(* CoDeSys 2.3.9.50 project: STP_PLC_arc.pro *)
(* Libraries: STANDARD.LIB 5.6.98 12:03:02 *)

(* Task configuration *)
TASK Standard (PRIORITY := 0, INTERVAL := T#10ms);
	STP
END_TASK

(* Global variable list: TwinCAT_Configuration *)
(* Generated automatically by TwinCAT - (read only) *)
VAR_CONFIG
	STP.LSL100A_MixerFloatSensor AT %IX276.0 : BOOL;	(*  ~ {LinkedWith:TIID^C6920 (EtherCAT)^ScadaRoom_KouplerUTP (EK1100)^ScadaRoom_KouplerFiber (EK1521)^InletWork_1(EK1501)^Term 5 (EL1809)^Channel 1^Input} *)
	STP.LSH100A_MixerFloatSensor AT %IX272.0 : BOOL;	(*  ~ {LinkedWith:TIID^C6920 (EtherCAT)^ScadaRoom_KouplerUTP (EK1100)^ScadaRoom_KouplerFiber (EK1521)^InletWork_1(EK1501)^Term 5 (EL1809)^Channel 2^Input} *)
	STP.LSH101A_EQFloatSensor AT %IX276.1 : BOOL;	(*  ~ {LinkedWith:TIID^C6920 (EtherCAT)^ScadaRoom_KouplerUTP (EK1100)^ScadaRoom_KouplerFiber (EK1521)^InletWork_1(EK1501)^Term 5 (EL1809)^Channel 3^Input} *)
	STP.LSHH101A_EQFloatSensor AT %IX276.2 : BOOL;	(*  ~ {LinkedWith:TIID^C6920 (EtherCAT)^ScadaRoom_KouplerUTP (EK1100)^ScadaRoom_KouplerFiber (EK1521)^InletWork_1(EK1501)^Term 5 (EL1809)^Channel 4^Input} *)
	STP.LSL101A_EQFloatSensor AT %IX256.1 : BOOL;	(*  ~ {LinkedWith:TIID^C6920 (EtherCAT)^ScadaRoom_KouplerUTP (EK1100)^ScadaRoom_KouplerFiber (EK1521)^InletWork_1(EK1501)^Term 5 (EL1809)^Channel 5^Input} *)
	STP.LSH105A1_StreamLineFlow AT %IX276.3 : BOOL;	(*  ~ {LinkedWith:TIID^C6920 (EtherCAT)^ScadaRoom_KouplerUTP (EK1100)^ScadaRoom_KouplerFiber (EK1521)^InletWork_1(EK1501)^Term 5 (EL1809)^Channel 6^Input} *)
	STP.LSHH105A2_StreamLineOverflow AT %IX276.4 : BOOL;	(*  ~ {LinkedWith:TIID^C6920 (EtherCAT)^ScadaRoom_KouplerUTP (EK1100)^ScadaRoom_KouplerFiber (EK1521)^InletWork_1(EK1501)^Term 5 (EL1809)^Channel 7^Input} *)
	STP.LSL103A_SBRFloatSensor AT %IX256.2 : BOOL;	(*  ~ {LinkedWith:TIID^C6920 (EtherCAT)^ScadaRoom_KouplerUTP (EK1100)^ScadaRoom_KouplerFiber (EK1521)^InletWork_1(EK1501)^Term 5 (EL1809)^Channel 8^Input} *)
	STP.LSHH103A_SBRFloatSensor AT %IX276.6 : BOOL;	(*  ~ {LinkedWith:TIID^C6920 (EtherCAT)^ScadaRoom_KouplerUTP (EK1100)^ScadaRoom_KouplerFiber (EK1521)^InletWork_1(EK1501)^Term 5 (EL1809)^Channel 9^Input} *)
	STP.LSH103A_SBRFloatSensor AT %IX276.5 : BOOL;	(*  ~ {LinkedWith:TIID^C6920 (EtherCAT)^ScadaRoom_KouplerUTP (EK1100)^ScadaRoom_KouplerFiber (EK1521)^InletWork_1(EK1501)^Term 5 (EL1809)^Channel 10^Input} *)
	STP.TMT01_FanStatus AT %IX276.7 : BOOL;	(*  ~ {LinkedWith:TIID^C6920 (EtherCAT)^ScadaRoom_KouplerUTP (EK1100)^ScadaRoom_KouplerFiber (EK1521)^InletWork_1(EK1501)^Term 5 (EL1809)^Channel 11^Input} *)
	STP.DP01_DoorPanelStatus AT %IX277.0 : BOOL;	(*  ~ {LinkedWith:TIID^C6920 (EtherCAT)^ScadaRoom_KouplerUTP (EK1100)^ScadaRoom_KouplerFiber (EK1521)^InletWork_1(EK1501)^Term 5 (EL1809)^Channel 12^Input} *)
	STP.LSD101A_EQFloatSensorDry AT %IX277.1 : BOOL;	(*  ~ {LinkedWith:TIID^C6920 (EtherCAT)^ScadaRoom_KouplerUTP (EK1100)^ScadaRoom_KouplerFiber (EK1521)^InletWork_1(EK1501)^Term 5 (EL1809)^Channel 13^Input} *)
	STP.LSD103A_SBRFloatSensorDry AT %IX277.2 : BOOL;	(*  ~ {LinkedWith:TIID^C6920 (EtherCAT)^ScadaRoom_KouplerUTP (EK1100)^ScadaRoom_KouplerFiber (EK1521)^InletWork_1(EK1501)^Term 5 (EL1809)^Channel 14^Input} *)
	STP.XV101A1_SolenoidValveSpray_OpenStat AT %IX277.3 : BOOL;	(*  ~ {LinkedWith:TIID^C6920 (EtherCAT)^ScadaRoom_KouplerUTP (EK1100)^ScadaRoom_KouplerFiber (EK1521)^InletWork_1(EK1501)^Term 6 (EL1809)^Channel 1^Input} *)
	STP.XV101A2_SolenoidValveSpray_OpenStat AT %IX277.4 : BOOL;	(*  ~ {LinkedWith:TIID^C6920 (EtherCAT)^ScadaRoom_KouplerUTP (EK1100)^ScadaRoom_KouplerFiber (EK1521)^InletWork_1(EK1501)^Term 6 (EL1809)^Channel 2^Input} *)
	STP.XV102A1_ContinuosValveWater_OpenStat AT %IX277.5 : BOOL;	(*  ~ {LinkedWith:TIID^C6920 (EtherCAT)^ScadaRoom_KouplerUTP (EK1100)^ScadaRoom_KouplerFiber (EK1521)^InletWork_1(EK1501)^Term 6 (EL1809)^Channel 3^Input} *)
	STP.XV100A1_GritRemovalValve_OpenStat AT %IX277.6 : BOOL;	(*  ~ {LinkedWith:TIID^C6920 (EtherCAT)^ScadaRoom_KouplerUTP (EK1100)^ScadaRoom_KouplerFiber (EK1521)^InletWork_1(EK1501)^Term 6 (EL1809)^Channel 5^Input} *)
	STP.XV100A2_GritRemovalValve_OpenStat AT %IX277.7 : BOOL;	(*  ~ {LinkedWith:TIID^C6920 (EtherCAT)^ScadaRoom_KouplerUTP (EK1100)^ScadaRoom_KouplerFiber (EK1521)^InletWork_1(EK1501)^Term 6 (EL1809)^Channel 6^Input} *)
	STP.PS101A1_Penstock_OpenStat AT %IX278.0 : BOOL;	(*  ~ {LinkedWith:TIID^C6920 (EtherCAT)^ScadaRoom_KouplerUTP (EK1100)^ScadaRoom_KouplerFiber (EK1521)^InletWork_1(EK1501)^Term 6 (EL1809)^Channel 7^Input} *)
	STP.PS101A2_Penstock_OpenStat AT %IX278.1 : BOOL;	(*  ~ {LinkedWith:TIID^C6920 (EtherCAT)^ScadaRoom_KouplerUTP (EK1100)^ScadaRoom_KouplerFiber (EK1521)^InletWork_1(EK1501)^Term 6 (EL1809)^Channel 8^Input} *)
	STP.PS101A1_Penstock_CloseStat AT %IX278.2 : BOOL;	(*  ~ {LinkedWith:TIID^C6920 (EtherCAT)^ScadaRoom_KouplerUTP (EK1100)^ScadaRoom_KouplerFiber (EK1521)^InletWork_1(EK1501)^Term 6 (EL1809)^Channel 9^Input} *)
	STP.PS101A2_Penstock_CloseStat AT %IX278.3 : BOOL;	(*  ~ {LinkedWith:TIID^C6920 (EtherCAT)^ScadaRoom_KouplerUTP (EK1100)^ScadaRoom_KouplerFiber (EK1521)^InletWork_1(EK1501)^Term 6 (EL1809)^Channel 10^Input} *)
	STP.XV101A1_SolenoidValveSpray_CloseStat AT %IX278.4 : BOOL;	(*  ~ {LinkedWith:TIID^C6920 (EtherCAT)^ScadaRoom_KouplerUTP (EK1100)^ScadaRoom_KouplerFiber (EK1521)^InletWork_1(EK1501)^Term 6 (EL1809)^Channel 11^Input} *)
	STP.XV101A2_SolenoidValveSpray_CloseStat AT %IX278.5 : BOOL;	(*  ~ {LinkedWith:TIID^C6920 (EtherCAT)^ScadaRoom_KouplerUTP (EK1100)^ScadaRoom_KouplerFiber (EK1521)^InletWork_1(EK1501)^Term 6 (EL1809)^Channel 12^Input} *)
	STP.XV102A1_ContinuosValveWater_CloseStat AT %IX278.6 : BOOL;	(*  ~ {LinkedWith:TIID^C6920 (EtherCAT)^ScadaRoom_KouplerUTP (EK1100)^ScadaRoom_KouplerFiber (EK1521)^InletWork_1(EK1501)^Term 6 (EL1809)^Channel 13^Input} *)
	STP.XV100A1_GritRemovalValve_CloseStat AT %IX278.7 : BOOL;	(*  ~ {LinkedWith:TIID^C6920 (EtherCAT)^ScadaRoom_KouplerUTP (EK1100)^ScadaRoom_KouplerFiber (EK1521)^InletWork_1(EK1501)^Term 6 (EL1809)^Channel 14^Input} *)
	STP.XV100A2_GritRemovalValve_CloseStat AT %IX279.0 : BOOL;	(*  ~ {LinkedWith:TIID^C6920 (EtherCAT)^ScadaRoom_KouplerUTP (EK1100)^ScadaRoom_KouplerFiber (EK1521)^InletWork_1(EK1501)^Term 6 (EL1809)^Channel 15^Input} *)
	STP.M101A1_EQMixer_OverloadStat AT %IX279.1 : BOOL;	(*  ~ {LinkedWith:TIID^C6920 (EtherCAT)^ScadaRoom_KouplerUTP (EK1100)^ScadaRoom_KouplerFiber (EK1521)^InletWork_1(EK1501)^Term 7 (EL1809)^Channel 1^Input} *)
	STP.M101A1_EQMixer_IncompleteStat AT %IX279.2 : BOOL;	(*  ~ {LinkedWith:TIID^C6920 (EtherCAT)^ScadaRoom_KouplerUTP (EK1100)^ScadaRoom_KouplerFiber (EK1521)^InletWork_1(EK1501)^Term 7 (EL1809)^Channel 2^Input} *)
	STP.M101A2_EQMixer_OverloadStat AT %IX279.3 : BOOL;	(*  ~ {LinkedWith:TIID^C6920 (EtherCAT)^ScadaRoom_KouplerUTP (EK1100)^ScadaRoom_KouplerFiber (EK1521)^InletWork_1(EK1501)^Term 7 (EL1809)^Channel 3^Input} *)
	STP.M101A2_EQMixer_IncompleteStat AT %IX279.4 : BOOL;	(*  ~ {LinkedWith:TIID^C6920 (EtherCAT)^ScadaRoom_KouplerUTP (EK1100)^ScadaRoom_KouplerFiber (EK1521)^InletWork_1(EK1501)^Term 7 (EL1809)^Channel 4^Input} *)
	STP.P101A1_EQPump_OverloadStat AT %IX4.0 : BOOL;	(*  ~ {LinkedWith:TIID^C6920 (EtherCAT)^ScadaRoom_KouplerUTP (EK1100)^ScadaRoom_KouplerFiber (EK1521)^InletWork_1(EK1501)^Term 7 (EL1809)^Channel 5^Input} *)
	STP.P101A1_EQPump_IncompleteStat AT %IX4.1 : BOOL;	(*  ~ {LinkedWith:TIID^C6920 (EtherCAT)^ScadaRoom_KouplerUTP (EK1100)^ScadaRoom_KouplerFiber (EK1521)^InletWork_1(EK1501)^Term 7 (EL1809)^Channel 6^Input} *)
	STP.P101A2_EQPump_OverloadStat AT %IX4.2 : BOOL;	(*  ~ {LinkedWith:TIID^C6920 (EtherCAT)^ScadaRoom_KouplerUTP (EK1100)^ScadaRoom_KouplerFiber (EK1521)^InletWork_1(EK1501)^Term 7 (EL1809)^Channel 7^Input} *)
	STP.P101A2_EQPump_IncompleteStat AT %IX4.3 : BOOL;	(*  ~ {LinkedWith:TIID^C6920 (EtherCAT)^ScadaRoom_KouplerUTP (EK1100)^ScadaRoom_KouplerFiber (EK1521)^InletWork_1(EK1501)^Term 7 (EL1809)^Channel 8^Input} *)
	STP.PS101A1_Penstock_TripStat AT %IX4.4 : BOOL;	(*  ~ {LinkedWith:TIID^C6920 (EtherCAT)^ScadaRoom_KouplerUTP (EK1100)^ScadaRoom_KouplerFiber (EK1521)^InletWork_1(EK1501)^Term 7 (EL1809)^Channel 9^Input} *)
	STP.PS101A2_Penstock_TripStat AT %IX4.5 : BOOL;	(*  ~ {LinkedWith:TIID^C6920 (EtherCAT)^ScadaRoom_KouplerUTP (EK1100)^ScadaRoom_KouplerFiber (EK1521)^InletWork_1(EK1501)^Term 7 (EL1809)^Channel 10^Input} *)
	STP.F101A1_FineScr_OverloadStat AT %IX4.6 : BOOL;	(*  ~ {LinkedWith:TIID^C6920 (EtherCAT)^ScadaRoom_KouplerUTP (EK1100)^ScadaRoom_KouplerFiber (EK1521)^InletWork_1(EK1501)^Term 8 (EL1809)^Channel 1^Input} *)
	STP.F101A2_FineScr_OverloadStat AT %IX4.7 : BOOL;	(*  ~ {LinkedWith:TIID^C6920 (EtherCAT)^ScadaRoom_KouplerUTP (EK1100)^ScadaRoom_KouplerFiber (EK1521)^InletWork_1(EK1501)^Term 8 (EL1809)^Channel 2^Input} *)
	STP.C102A_ScreeningConveyer_OverloadStat AT %IX5.0 : BOOL;	(*  ~ {LinkedWith:TIID^C6920 (EtherCAT)^ScadaRoom_KouplerUTP (EK1100)^ScadaRoom_KouplerFiber (EK1521)^InletWork_1(EK1501)^Term 8 (EL1809)^Channel 3^Input} *)
	STP.C101A_ScreeningCompactor_OverloadStat AT %IX5.1 : BOOL;	(*  ~ {LinkedWith:TIID^C6920 (EtherCAT)^ScadaRoom_KouplerUTP (EK1100)^ScadaRoom_KouplerFiber (EK1521)^InletWork_1(EK1501)^Term 8 (EL1809)^Channel 4^Input} *)
	STP.C103A_GritClassifier_OverloadStat AT %IX5.2 : BOOL;	(*  ~ {LinkedWith:TIID^C6920 (EtherCAT)^ScadaRoom_KouplerUTP (EK1100)^ScadaRoom_KouplerFiber (EK1521)^InletWork_1(EK1501)^Term 8 (EL1809)^Channel 5^Input} *)
	STP.P102A1_SBRTransferPump_OverloadStat AT %IX5.3 : BOOL;	(*  ~ {LinkedWith:TIID^C6920 (EtherCAT)^ScadaRoom_KouplerUTP (EK1100)^ScadaRoom_KouplerFiber (EK1521)^InletWork_1(EK1501)^Term 8 (EL1809)^Channel 6^Input} *)
	STP.P102A1_SBRTransferPump_IncompleteStat AT %IX5.4 : BOOL;	(*  ~ {LinkedWith:TIID^C6920 (EtherCAT)^ScadaRoom_KouplerUTP (EK1100)^ScadaRoom_KouplerFiber (EK1521)^InletWork_1(EK1501)^Term 8 (EL1809)^Channel 7^Input} *)
	STP.P102A2_SBRTransferPump_OverloadStat AT %IX5.5 : BOOL;	(*  ~ {LinkedWith:TIID^C6920 (EtherCAT)^ScadaRoom_KouplerUTP (EK1100)^ScadaRoom_KouplerFiber (EK1521)^InletWork_1(EK1501)^Term 8 (EL1809)^Channel 8^Input} *)
	STP.P102A2_SBRTransferPump_IncompleteStat AT %IX5.6 : BOOL;	(*  ~ {LinkedWith:TIID^C6920 (EtherCAT)^ScadaRoom_KouplerUTP (EK1100)^ScadaRoom_KouplerFiber (EK1521)^InletWork_1(EK1501)^Term 8 (EL1809)^Channel 9^Input} *)
	STP.M101A1_EQMixer_LocalRemoteStat AT %IX5.7 : BOOL;	(*  ~ {LinkedWith:TIID^C6920 (EtherCAT)^ScadaRoom_KouplerUTP (EK1100)^ScadaRoom_KouplerFiber (EK1521)^InletWork_1(EK1501)^Term 9 (EL1809)^Channel 1^Input} *)
	STP.M101A2_EQMixer_LocalRemoteStat AT %IX6.0 : BOOL;	(*  ~ {LinkedWith:TIID^C6920 (EtherCAT)^ScadaRoom_KouplerUTP (EK1100)^ScadaRoom_KouplerFiber (EK1521)^InletWork_1(EK1501)^Term 9 (EL1809)^Channel 2^Input} *)
	STP.P101A1_EQPump_LocalRemoteStat AT %IX6.1 : BOOL;	(*  ~ {LinkedWith:TIID^C6920 (EtherCAT)^ScadaRoom_KouplerUTP (EK1100)^ScadaRoom_KouplerFiber (EK1521)^InletWork_1(EK1501)^Term 9 (EL1809)^Channel 3^Input} *)
	STP.P101A2_EQPump_LocalRemoteStat AT %IX6.2 : BOOL;	(*  ~ {LinkedWith:TIID^C6920 (EtherCAT)^ScadaRoom_KouplerUTP (EK1100)^ScadaRoom_KouplerFiber (EK1521)^InletWork_1(EK1501)^Term 9 (EL1809)^Channel 4^Input} *)
	STP.F101A1_FineScr_LocalRemoteStat AT %IX6.3 : BOOL;	(*  ~ {LinkedWith:TIID^C6920 (EtherCAT)^ScadaRoom_KouplerUTP (EK1100)^ScadaRoom_KouplerFiber (EK1521)^InletWork_1(EK1501)^Term 9 (EL1809)^Channel 5^Input} *)
	STP.F101A2_FineScr_LocalRemoteStat AT %IX6.4 : BOOL;	(*  ~ {LinkedWith:TIID^C6920 (EtherCAT)^ScadaRoom_KouplerUTP (EK1100)^ScadaRoom_KouplerFiber (EK1521)^InletWork_1(EK1501)^Term 9 (EL1809)^Channel 6^Input} *)
	STP.C102A_ScreenConveyer_LocalRemoteStat AT %IX6.5 : BOOL;	(*  ~ {LinkedWith:TIID^C6920 (EtherCAT)^ScadaRoom_KouplerUTP (EK1100)^ScadaRoom_KouplerFiber (EK1521)^InletWork_1(EK1501)^Term 9 (EL1809)^Channel 7^Input} *)
	STP.C101A_ScreenCompactor_LocalRemoteStat AT %IX6.6 : BOOL;	(*  ~ {LinkedWith:TIID^C6920 (EtherCAT)^ScadaRoom_KouplerUTP (EK1100)^ScadaRoom_KouplerFiber (EK1521)^InletWork_1(EK1501)^Term 9 (EL1809)^Channel 8^Input} *)
	STP.C103A_GritClasifier_LocalRemoteStat AT %IX6.7 : BOOL;	(*  ~ {LinkedWith:TIID^C6920 (EtherCAT)^ScadaRoom_KouplerUTP (EK1100)^ScadaRoom_KouplerFiber (EK1521)^InletWork_1(EK1501)^Term 9 (EL1809)^Channel 9^Input} *)
	STP.P102A1_SBRTransferPump_LocalRemoteStat AT %IX7.0 : BOOL;	(*  ~ {LinkedWith:TIID^C6920 (EtherCAT)^ScadaRoom_KouplerUTP (EK1100)^ScadaRoom_KouplerFiber (EK1521)^InletWork_1(EK1501)^Term 9 (EL1809)^Channel 10^Input} *)
	STP.P102A2_SBRTransferPump_LocalRemoteStat AT %IX7.1 : BOOL;	(*  ~ {LinkedWith:TIID^C6920 (EtherCAT)^ScadaRoom_KouplerUTP (EK1100)^ScadaRoom_KouplerFiber (EK1521)^InletWork_1(EK1501)^Term 9 (EL1809)^Channel 11^Input} *)
	STP.PS101A1_Penstock_LocalRemoteStat AT %IX296.0 : BOOL;	(*  ~ {LinkedWith:TIID^C6920 (EtherCAT)^ScadaRoom_KouplerUTP (EK1100)^ScadaRoom_KouplerFiber (EK1521)^InletWork_1(EK1501)^Term 10 (EL1809)^Channel 12^Input} *)
	STP.PS101A2_Penstock_LocalRemoteStat AT %IX296.1 : BOOL;	(*  ~ {LinkedWith:TIID^C6920 (EtherCAT)^ScadaRoom_KouplerUTP (EK1100)^ScadaRoom_KouplerFiber (EK1521)^InletWork_1(EK1501)^Term 10 (EL1809)^Channel 13^Input} *)
	STP.M101A1_EQMixer_RunStat AT %IX7.2 : BOOL;	(*  ~ {LinkedWith:TIID^C6920 (EtherCAT)^ScadaRoom_KouplerUTP (EK1100)^ScadaRoom_KouplerFiber (EK1521)^InletWork_1(EK1501)^Term 10 (EL1809)^Channel 1^Input} *)
	STP.M101A2_EQMixer_RunStat AT %IX7.3 : BOOL;	(*  ~ {LinkedWith:TIID^C6920 (EtherCAT)^ScadaRoom_KouplerUTP (EK1100)^ScadaRoom_KouplerFiber (EK1521)^InletWork_1(EK1501)^Term 10 (EL1809)^Channel 2^Input} *)
	STP.P101A1_EQPump_RunStat AT %IX7.4 : BOOL;	(*  ~ {LinkedWith:TIID^C6920 (EtherCAT)^ScadaRoom_KouplerUTP (EK1100)^ScadaRoom_KouplerFiber (EK1521)^InletWork_1(EK1501)^Term 10 (EL1809)^Channel 3^Input} *)
	STP.P101A2_EQPump_RunStat AT %IX7.5 : BOOL;	(*  ~ {LinkedWith:TIID^C6920 (EtherCAT)^ScadaRoom_KouplerUTP (EK1100)^ScadaRoom_KouplerFiber (EK1521)^InletWork_1(EK1501)^Term 10 (EL1809)^Channel 4^Input} *)
	STP.F101A1_FineScr_RunStat AT %IX7.6 : BOOL;	(*  ~ {LinkedWith:TIID^C6920 (EtherCAT)^ScadaRoom_KouplerUTP (EK1100)^ScadaRoom_KouplerFiber (EK1521)^InletWork_1(EK1501)^Term 10 (EL1809)^Channel 5^Input} *)
	STP.F101A2_FineScr_RunStat AT %IX7.7 : BOOL;	(*  ~ {LinkedWith:TIID^C6920 (EtherCAT)^ScadaRoom_KouplerUTP (EK1100)^ScadaRoom_KouplerFiber (EK1521)^InletWork_1(EK1501)^Term 10 (EL1809)^Channel 6^Input} *)
	STP.C102A_ScreenConveyer_RunStat AT %IX8.0 : BOOL;	(*  ~ {LinkedWith:TIID^C6920 (EtherCAT)^ScadaRoom_KouplerUTP (EK1100)^ScadaRoom_KouplerFiber (EK1521)^InletWork_1(EK1501)^Term 10 (EL1809)^Channel 7^Input} *)
	STP.C101A_ScreenCompactor_RunStat AT %IX8.1 : BOOL;	(*  ~ {LinkedWith:TIID^C6920 (EtherCAT)^ScadaRoom_KouplerUTP (EK1100)^ScadaRoom_KouplerFiber (EK1521)^InletWork_1(EK1501)^Term 10 (EL1809)^Channel 8^Input} *)
	STP.C103A_GritClasifier_RunStat AT %IX8.2 : BOOL;	(*  ~ {LinkedWith:TIID^C6920 (EtherCAT)^ScadaRoom_KouplerUTP (EK1100)^ScadaRoom_KouplerFiber (EK1521)^InletWork_1(EK1501)^Term 10 (EL1809)^Channel 9^Input} *)
	STP.P102A1_SBRTransferPump_RunStat AT %IX8.3 : BOOL;	(*  ~ {LinkedWith:TIID^C6920 (EtherCAT)^ScadaRoom_KouplerUTP (EK1100)^ScadaRoom_KouplerFiber (EK1521)^InletWork_1(EK1501)^Term 10 (EL1809)^Channel 10^Input} *)
	STP.P102A2_SBRTransferPump_RunStat AT %IX8.4 : BOOL;	(*  ~ {LinkedWith:TIID^C6920 (EtherCAT)^ScadaRoom_KouplerUTP (EK1100)^ScadaRoom_KouplerFiber (EK1521)^InletWork_1(EK1501)^Term 10 (EL1809)^Channel 11^Input} *)
	STP.M101A1_EQMixer_EStopStat AT %IX8.5 : BOOL;	(*  ~ {LinkedWith:TIID^C6920 (EtherCAT)^ScadaRoom_KouplerUTP (EK1100)^ScadaRoom_KouplerFiber (EK1521)^InletWork_1(EK1501)^Term 11 (EL1809)^Channel 1^Input} *)
	STP.M101A2_EQMixer_EStopStat AT %IX8.6 : BOOL;	(*  ~ {LinkedWith:TIID^C6920 (EtherCAT)^ScadaRoom_KouplerUTP (EK1100)^ScadaRoom_KouplerFiber (EK1521)^InletWork_1(EK1501)^Term 11 (EL1809)^Channel 2^Input} *)
	STP.P101A1_EQPump_EStopStat AT %IX8.7 : BOOL;	(*  ~ {LinkedWith:TIID^C6920 (EtherCAT)^ScadaRoom_KouplerUTP (EK1100)^ScadaRoom_KouplerFiber (EK1521)^InletWork_1(EK1501)^Term 11 (EL1809)^Channel 3^Input} *)
	STP.P101A2_EQPump_EStopStat AT %IX9.0 : BOOL;	(*  ~ {LinkedWith:TIID^C6920 (EtherCAT)^ScadaRoom_KouplerUTP (EK1100)^ScadaRoom_KouplerFiber (EK1521)^InletWork_1(EK1501)^Term 11 (EL1809)^Channel 4^Input} *)
	STP.F101A1_FineScr_EStopStat AT %IX9.1 : BOOL;	(*  ~ {LinkedWith:TIID^C6920 (EtherCAT)^ScadaRoom_KouplerUTP (EK1100)^ScadaRoom_KouplerFiber (EK1521)^InletWork_1(EK1501)^Term 11 (EL1809)^Channel 5^Input} *)
	STP.F101A2_FineScr_EStopStat AT %IX9.2 : BOOL;	(*  ~ {LinkedWith:TIID^C6920 (EtherCAT)^ScadaRoom_KouplerUTP (EK1100)^ScadaRoom_KouplerFiber (EK1521)^InletWork_1(EK1501)^Term 11 (EL1809)^Channel 6^Input} *)
	STP.C102A_ScreenConveyer_EStopStat AT %IX9.3 : BOOL;	(*  ~ {LinkedWith:TIID^C6920 (EtherCAT)^ScadaRoom_KouplerUTP (EK1100)^ScadaRoom_KouplerFiber (EK1521)^InletWork_1(EK1501)^Term 11 (EL1809)^Channel 7^Input} *)
	STP.C101A_ScreenCompactor_EStopStat AT %IX9.4 : BOOL;	(*  ~ {LinkedWith:TIID^C6920 (EtherCAT)^ScadaRoom_KouplerUTP (EK1100)^ScadaRoom_KouplerFiber (EK1521)^InletWork_1(EK1501)^Term 11 (EL1809)^Channel 8^Input} *)
	STP.C103A_GritClasifier_EStopStat AT %IX9.5 : BOOL;	(*  ~ {LinkedWith:TIID^C6920 (EtherCAT)^ScadaRoom_KouplerUTP (EK1100)^ScadaRoom_KouplerFiber (EK1521)^InletWork_1(EK1501)^Term 11 (EL1809)^Channel 9^Input} *)
	STP.P102A1_SBRTransferPump_EStopStat AT %IX9.6 : BOOL;	(*  ~ {LinkedWith:TIID^C6920 (EtherCAT)^ScadaRoom_KouplerUTP (EK1100)^ScadaRoom_KouplerFiber (EK1521)^InletWork_1(EK1501)^Term 11 (EL1809)^Channel 10^Input} *)
	STP.P102A2_SBRTransferPump_EStopStat AT %IX9.7 : BOOL;	(*  ~ {LinkedWith:TIID^C6920 (EtherCAT)^ScadaRoom_KouplerUTP (EK1100)^ScadaRoom_KouplerFiber (EK1521)^InletWork_1(EK1501)^Term 11 (EL1809)^Channel 11^Input} *)
	STP.B101A1_AirBlower_OverloadStat AT %IX10.0 : BOOL;	(*  ~ {LinkedWith:TIID^C6920 (EtherCAT)^ScadaRoom_KouplerUTP (EK1100)^ScadaRoom_KouplerFiber (EK1521)^InletWork_1(EK1501)^Term 12 (EL1809)^Channel 1^Input} *)
	STP.B101A1_AirBlower_IncompleteStat AT %IX10.1 : BOOL;	(*  ~ {LinkedWith:TIID^C6920 (EtherCAT)^ScadaRoom_KouplerUTP (EK1100)^ScadaRoom_KouplerFiber (EK1521)^InletWork_1(EK1501)^Term 12 (EL1809)^Channel 2^Input} *)
	STP.B101A2_AirBlower_OverloadStat AT %IX10.2 : BOOL;	(*  ~ {LinkedWith:TIID^C6920 (EtherCAT)^ScadaRoom_KouplerUTP (EK1100)^ScadaRoom_KouplerFiber (EK1521)^InletWork_1(EK1501)^Term 12 (EL1809)^Channel 3^Input} *)
	STP.B101A2_AirBlower_IncompleteStat AT %IX10.3 : BOOL;	(*  ~ {LinkedWith:TIID^C6920 (EtherCAT)^ScadaRoom_KouplerUTP (EK1100)^ScadaRoom_KouplerFiber (EK1521)^InletWork_1(EK1501)^Term 12 (EL1809)^Channel 4^Input} *)
	STP.B101A1_AirBlower_LocalRemoteStat AT %IX10.4 : BOOL;	(*  ~ {LinkedWith:TIID^C6920 (EtherCAT)^ScadaRoom_KouplerUTP (EK1100)^ScadaRoom_KouplerFiber (EK1521)^InletWork_1(EK1501)^Term 12 (EL1809)^Channel 5^Input} *)
	STP.B101A2_AirBlower_LocalRemoteStat AT %IX10.5 : BOOL;	(*  ~ {LinkedWith:TIID^C6920 (EtherCAT)^ScadaRoom_KouplerUTP (EK1100)^ScadaRoom_KouplerFiber (EK1521)^InletWork_1(EK1501)^Term 12 (EL1809)^Channel 6^Input} *)
	STP.B101A1_AirBlower_OnOffStat AT %IX10.6 : BOOL;	(*  ~ {LinkedWith:TIID^C6920 (EtherCAT)^ScadaRoom_KouplerUTP (EK1100)^ScadaRoom_KouplerFiber (EK1521)^InletWork_1(EK1501)^Term 12 (EL1809)^Channel 7^Input} *)
	STP.B101A2_AirBlower_OnOffStat AT %IX10.7 : BOOL;	(*  ~ {LinkedWith:TIID^C6920 (EtherCAT)^ScadaRoom_KouplerUTP (EK1100)^ScadaRoom_KouplerFiber (EK1521)^InletWork_1(EK1501)^Term 12 (EL1809)^Channel 8^Input} *)
	STP.B101A1_AirBlower_EStopStat AT %IX11.0 : BOOL;	(*  ~ {LinkedWith:TIID^C6920 (EtherCAT)^ScadaRoom_KouplerUTP (EK1100)^ScadaRoom_KouplerFiber (EK1521)^InletWork_1(EK1501)^Term 12 (EL1809)^Channel 9^Input} *)
	STP.B101A2_AirBlower_EStopStat AT %IX11.1 : BOOL;	(*  ~ {LinkedWith:TIID^C6920 (EtherCAT)^ScadaRoom_KouplerUTP (EK1100)^ScadaRoom_KouplerFiber (EK1521)^InletWork_1(EK1501)^Term 12 (EL1809)^Channel 10^Input} *)
	STP.XV101A1_SolenoidValveSpray_OpenCmd AT %QX0.0 : BOOL;	(*  ~ {LinkedWith:TIID^C6920 (EtherCAT)^ScadaRoom_KouplerUTP (EK1100)^ScadaRoom_KouplerFiber (EK1521)^InletWork_1(EK1501)^Term 13 (EL2809)^Channel 1^Output} *)
	STP.XV101A2_SolenoidValveSpray_OpenCmd AT %QX0.1 : BOOL;	(*  ~ {LinkedWith:TIID^C6920 (EtherCAT)^ScadaRoom_KouplerUTP (EK1100)^ScadaRoom_KouplerFiber (EK1521)^InletWork_1(EK1501)^Term 13 (EL2809)^Channel 2^Output} *)
	STP.XV102A1_ContinuosValveWater_OpenCmd AT %QX0.2 : BOOL;	(*  ~ {LinkedWith:TIID^C6920 (EtherCAT)^ScadaRoom_KouplerUTP (EK1100)^ScadaRoom_KouplerFiber (EK1521)^InletWork_1(EK1501)^Term 13 (EL2809)^Channel 3^Output} *)
	STP.F101A1_FineScr_RunCmd AT %QX0.4 : BOOL;	(*  ~ {LinkedWith:TIID^C6920 (EtherCAT)^ScadaRoom_KouplerUTP (EK1100)^ScadaRoom_KouplerFiber (EK1521)^InletWork_1(EK1501)^Term 13 (EL2809)^Channel 5^Output} *)
	STP.F101A2_FineScr_RunCmd AT %QX0.5 : BOOL;	(*  ~ {LinkedWith:TIID^C6920 (EtherCAT)^ScadaRoom_KouplerUTP (EK1100)^ScadaRoom_KouplerFiber (EK1521)^InletWork_1(EK1501)^Term 13 (EL2809)^Channel 6^Output} *)
	STP.C102A_ScreenConveyer_RunCmd AT %QX0.6 : BOOL;	(*  ~ {LinkedWith:TIID^C6920 (EtherCAT)^ScadaRoom_KouplerUTP (EK1100)^ScadaRoom_KouplerFiber (EK1521)^InletWork_1(EK1501)^Term 13 (EL2809)^Channel 7^Output} *)
	STP.C101A_ScreenCompactor_RunCmd AT %QX68.0 : BOOL;	(*  ~ {LinkedWith:TIID^C6920 (EtherCAT)^ScadaRoom_KouplerUTP (EK1100)^ScadaRoom_KouplerFiber (EK1521)^InletWork_1(EK1501)^Term 13 (EL2809)^Channel 8^Output} *)
	STP.C103A_GritClasifier_RunCmd AT %QX1.0 : BOOL;	(*  ~ {LinkedWith:TIID^C6920 (EtherCAT)^ScadaRoom_KouplerUTP (EK1100)^ScadaRoom_KouplerFiber (EK1521)^InletWork_1(EK1501)^Term 13 (EL2809)^Channel 9^Output} *)
	STP.PS101A1_Penstock_OpenCmd AT %QX1.1 : BOOL;	(*  ~ {LinkedWith:TIID^C6920 (EtherCAT)^ScadaRoom_KouplerUTP (EK1100)^ScadaRoom_KouplerFiber (EK1521)^InletWork_1(EK1501)^Term 13 (EL2809)^Channel 10^Output} *)
	STP.PS101A1_Penstock_CloseCmd AT %QX1.2 : BOOL;	(*  ~ {LinkedWith:TIID^C6920 (EtherCAT)^ScadaRoom_KouplerUTP (EK1100)^ScadaRoom_KouplerFiber (EK1521)^InletWork_1(EK1501)^Term 13 (EL2809)^Channel 11^Output} *)
	STP.PS101A2_Penstock_OpenCmd AT %QX1.3 : BOOL;	(*  ~ {LinkedWith:TIID^C6920 (EtherCAT)^ScadaRoom_KouplerUTP (EK1100)^ScadaRoom_KouplerFiber (EK1521)^InletWork_1(EK1501)^Term 13 (EL2809)^Channel 12^Output} *)
	STP.PS101A2_Penstock_CloseCmd AT %QX1.4 : BOOL;	(*  ~ {LinkedWith:TIID^C6920 (EtherCAT)^ScadaRoom_KouplerUTP (EK1100)^ScadaRoom_KouplerFiber (EK1521)^InletWork_1(EK1501)^Term 13 (EL2809)^Channel 13^Output} *)
	STP.XV100A1_GritRemovalValve_OpenCmd AT %QX1.5 : BOOL;	(*  ~ {LinkedWith:TIID^C6920 (EtherCAT)^ScadaRoom_KouplerUTP (EK1100)^ScadaRoom_KouplerFiber (EK1521)^InletWork_1(EK1501)^Term 13 (EL2809)^Channel 14^Output} *)
	STP.XV100A2_GritRemovalValve_OpenCmd AT %QX1.6 : BOOL;	(*  ~ {LinkedWith:TIID^C6920 (EtherCAT)^ScadaRoom_KouplerUTP (EK1100)^ScadaRoom_KouplerFiber (EK1521)^InletWork_1(EK1501)^Term 13 (EL2809)^Channel 15^Output} *)
	STP.P101A1_EQPump_RunCmd AT %QX1.7 : BOOL;	(*  ~ {LinkedWith:TIID^C6920 (EtherCAT)^ScadaRoom_KouplerUTP (EK1100)^ScadaRoom_KouplerFiber (EK1521)^InletWork_1(EK1501)^Term 14 (EL2809)^Channel 1^Output} *)
	STP.P101A2_EQPump_RunCmd AT %QX2.0 : BOOL;	(*  ~ {LinkedWith:TIID^C6920 (EtherCAT)^ScadaRoom_KouplerUTP (EK1100)^ScadaRoom_KouplerFiber (EK1521)^InletWork_1(EK1501)^Term 14 (EL2809)^Channel 2^Output} *)
	STP.M101A1_EQMixer_RunCmd AT %QX2.1 : BOOL;	(*  ~ {LinkedWith:TIID^C6920 (EtherCAT)^ScadaRoom_KouplerUTP (EK1100)^ScadaRoom_KouplerFiber (EK1521)^InletWork_1(EK1501)^Term 14 (EL2809)^Channel 3^Output} *)
	STP.M101A2_EQMixer_RunCmd AT %QX2.2 : BOOL;	(*  ~ {LinkedWith:TIID^C6920 (EtherCAT)^ScadaRoom_KouplerUTP (EK1100)^ScadaRoom_KouplerFiber (EK1521)^InletWork_1(EK1501)^Term 14 (EL2809)^Channel 4^Output} *)
	STP.B101A1_AirBlower_RunCmd AT %QX2.3 : BOOL;	(*  ~ {LinkedWith:TIID^C6920 (EtherCAT)^ScadaRoom_KouplerUTP (EK1100)^ScadaRoom_KouplerFiber (EK1521)^InletWork_1(EK1501)^Term 14 (EL2809)^Channel 5^Output} *)
	STP.B101A2_AirBlower_RunCmd AT %QX2.4 : BOOL;	(*  ~ {LinkedWith:TIID^C6920 (EtherCAT)^ScadaRoom_KouplerUTP (EK1100)^ScadaRoom_KouplerFiber (EK1521)^InletWork_1(EK1501)^Term 14 (EL2809)^Channel 6^Output} *)
	STP.P102A1_SBRTransferPump_RunCmd AT %QX2.5 : BOOL;	(*  ~ {LinkedWith:TIID^C6920 (EtherCAT)^ScadaRoom_KouplerUTP (EK1100)^ScadaRoom_KouplerFiber (EK1521)^InletWork_1(EK1501)^Term 14 (EL2809)^Channel 7^Output} *)
	STP.P102A2_SBRTransferPump_RunCmd AT %QX2.6 : BOOL;	(*  ~ {LinkedWith:TIID^C6920 (EtherCAT)^ScadaRoom_KouplerUTP (EK1100)^ScadaRoom_KouplerFiber (EK1521)^InletWork_1(EK1501)^Term 14 (EL2809)^Channel 8^Output} *)
	STP.AUX101A_EQFloatSensor_AlarmS1 AT %QX2.7 : BOOL;	(*  ~ {LinkedWith:TIID^C6920 (EtherCAT)^ScadaRoom_KouplerUTP (EK1100)^ScadaRoom_KouplerFiber (EK1521)^InletWork_1(EK1501)^Term 14 (EL2809)^Channel 9^Output} *)
	STP.AUX104A_SBRFloatSensor_AlarmS1 AT %QX3.0 : BOOL;	(*  ~ {LinkedWith:TIID^C6920 (EtherCAT)^ScadaRoom_KouplerUTP (EK1100)^ScadaRoom_KouplerFiber (EK1521)^InletWork_1(EK1501)^Term 14 (EL2809)^Channel 10^Output} *)
	STP.AUX105A_StreamSensorOverflow_AlarmS1 AT %QX3.1 : BOOL;	(*  ~ {LinkedWith:TIID^C6920 (EtherCAT)^ScadaRoom_KouplerUTP (EK1100)^ScadaRoom_KouplerFiber (EK1521)^InletWork_1(EK1501)^Term 14 (EL2809)^Channel 11^Output} *)
	STP.AUX101_CommonAlarm AT %QX72.0 : BOOL;	(*  ~ {LinkedWith:TIID^C6920 (EtherCAT)^ScadaRoom_KouplerUTP (EK1100)^ScadaRoom_KouplerFiber (EK1521)^InletWork_1(EK1501)^Term 14 (EL2809)^Channel 12^Output} *)
	STP.AUX102_PLCRunStat AT %QX72.1 : BOOL;	(*  ~ {LinkedWith:TIID^C6920 (EtherCAT)^ScadaRoom_KouplerUTP (EK1100)^ScadaRoom_KouplerFiber (EK1521)^InletWork_1(EK1501)^Term 14 (EL2809)^Channel 13^Output} *)
	STP.LSL100B_MixerFloatSensor AT %IX11.2 : BOOL;	(*  ~ {LinkedWith:TIID^C6920 (EtherCAT)^ScadaRoom_KouplerUTP (EK1100)^ScadaRoom_KouplerFiber (EK1521)^InletWork_1(EK1501)^InletWork_2 (EK1122)^Term 16 (EK1100)^Term 17 (EL1809)^Channel 1^Input} *)
	STP.LSH100B_MixerFloatSensor AT %IX256.3 : BOOL;	(*  ~ {LinkedWith:TIID^C6920 (EtherCAT)^ScadaRoom_KouplerUTP (EK1100)^ScadaRoom_KouplerFiber (EK1521)^InletWork_1(EK1501)^InletWork_2 (EK1122)^Term 16 (EK1100)^Term 17 (EL1809)^Channel 2^Input} *)
	STP.LSH101B_EQFloatSensor AT %IX11.4 : BOOL;	(*  ~ {LinkedWith:TIID^C6920 (EtherCAT)^ScadaRoom_KouplerUTP (EK1100)^ScadaRoom_KouplerFiber (EK1521)^InletWork_1(EK1501)^InletWork_2 (EK1122)^Term 16 (EK1100)^Term 17 (EL1809)^Channel 3^Input} *)
	STP.LSHH101B_EQFloatSensor AT %IX11.5 : BOOL;	(*  ~ {LinkedWith:TIID^C6920 (EtherCAT)^ScadaRoom_KouplerUTP (EK1100)^ScadaRoom_KouplerFiber (EK1521)^InletWork_1(EK1501)^InletWork_2 (EK1122)^Term 16 (EK1100)^Term 17 (EL1809)^Channel 4^Input} *)
	STP.LSL101B_EQFloatSensor AT %IX256.4 : BOOL;	(*  ~ {LinkedWith:TIID^C6920 (EtherCAT)^ScadaRoom_KouplerUTP (EK1100)^ScadaRoom_KouplerFiber (EK1521)^InletWork_1(EK1501)^InletWork_2 (EK1122)^Term 16 (EK1100)^Term 17 (EL1809)^Channel 5^Input} *)
	STP.LSH105B1_StreamLineFlow AT %IX11.7 : BOOL;	(*  ~ {LinkedWith:TIID^C6920 (EtherCAT)^ScadaRoom_KouplerUTP (EK1100)^ScadaRoom_KouplerFiber (EK1521)^InletWork_1(EK1501)^InletWork_2 (EK1122)^Term 16 (EK1100)^Term 17 (EL1809)^Channel 6^Input} *)
	STP.LSHH105B2_StreamLineOverflow AT %IX12.0 : BOOL;	(*  ~ {LinkedWith:TIID^C6920 (EtherCAT)^ScadaRoom_KouplerUTP (EK1100)^ScadaRoom_KouplerFiber (EK1521)^InletWork_1(EK1501)^InletWork_2 (EK1122)^Term 16 (EK1100)^Term 17 (EL1809)^Channel 7^Input} *)
	STP.LSH103B_SBRFloatSensor AT %IX12.1 : BOOL;	(*  ~ {LinkedWith:TIID^C6920 (EtherCAT)^ScadaRoom_KouplerUTP (EK1100)^ScadaRoom_KouplerFiber (EK1521)^InletWork_1(EK1501)^InletWork_2 (EK1122)^Term 16 (EK1100)^Term 17 (EL1809)^Channel 8^Input} *)
	STP.LSHH103B_SBRFloatSensor AT %IX12.2 : BOOL;	(*  ~ {LinkedWith:TIID^C6920 (EtherCAT)^ScadaRoom_KouplerUTP (EK1100)^ScadaRoom_KouplerFiber (EK1521)^InletWork_1(EK1501)^InletWork_2 (EK1122)^Term 16 (EK1100)^Term 17 (EL1809)^Channel 9^Input} *)
	STP.LSL103B_SBRFloatSensor AT %IX256.5 : BOOL;	(*  ~ {LinkedWith:TIID^C6920 (EtherCAT)^ScadaRoom_KouplerUTP (EK1100)^ScadaRoom_KouplerFiber (EK1521)^InletWork_1(EK1501)^InletWork_2 (EK1122)^Term 16 (EK1100)^Term 17 (EL1809)^Channel 10^Input} *)
	STP.LSD101B_EQFloatSensorDry AT %IX12.4 : BOOL;	(*  ~ {LinkedWith:TIID^C6920 (EtherCAT)^ScadaRoom_KouplerUTP (EK1100)^ScadaRoom_KouplerFiber (EK1521)^InletWork_1(EK1501)^InletWork_2 (EK1122)^Term 16 (EK1100)^Term 17 (EL1809)^Channel 11^Input} *)
	STP.LSD103B_SBRFloatSensorDry AT %IX12.5 : BOOL;	(*  ~ {LinkedWith:TIID^C6920 (EtherCAT)^ScadaRoom_KouplerUTP (EK1100)^ScadaRoom_KouplerFiber (EK1521)^InletWork_1(EK1501)^InletWork_2 (EK1122)^Term 16 (EK1100)^Term 17 (EL1809)^Channel 12^Input} *)
	STP.XV101B1_SolenoidValveSpray_OpenStat AT %IX12.6 : BOOL;	(*  ~ {LinkedWith:TIID^C6920 (EtherCAT)^ScadaRoom_KouplerUTP (EK1100)^ScadaRoom_KouplerFiber (EK1521)^InletWork_1(EK1501)^InletWork_2 (EK1122)^Term 16 (EK1100)^Term 18 (EL1809)^Channel 1^Input} *)
	STP.XV101B2_SolenoidValveSpray_OpenStat AT %IX12.7 : BOOL;	(*  ~ {LinkedWith:TIID^C6920 (EtherCAT)^ScadaRoom_KouplerUTP (EK1100)^ScadaRoom_KouplerFiber (EK1521)^InletWork_1(EK1501)^InletWork_2 (EK1122)^Term 16 (EK1100)^Term 18 (EL1809)^Channel 2^Input} *)
	STP.XV102B1_ContinuosValveWater_OpenStat AT %IX13.0 : BOOL;	(*  ~ {LinkedWith:TIID^C6920 (EtherCAT)^ScadaRoom_KouplerUTP (EK1100)^ScadaRoom_KouplerFiber (EK1521)^InletWork_1(EK1501)^InletWork_2 (EK1122)^Term 16 (EK1100)^Term 18 (EL1809)^Channel 3^Input} *)
	STP.XV100B1_GritRemovalValve_OpenStat AT %IX13.1 : BOOL;	(*  ~ {LinkedWith:TIID^C6920 (EtherCAT)^ScadaRoom_KouplerUTP (EK1100)^ScadaRoom_KouplerFiber (EK1521)^InletWork_1(EK1501)^InletWork_2 (EK1122)^Term 16 (EK1100)^Term 18 (EL1809)^Channel 5^Input} *)
	STP.XV100B2_GritRemovalValve_OpenStat AT %IX13.2 : BOOL;	(*  ~ {LinkedWith:TIID^C6920 (EtherCAT)^ScadaRoom_KouplerUTP (EK1100)^ScadaRoom_KouplerFiber (EK1521)^InletWork_1(EK1501)^InletWork_2 (EK1122)^Term 16 (EK1100)^Term 18 (EL1809)^Channel 6^Input} *)
	STP.PS101B1_Penstock_OpenStat AT %IX13.3 : BOOL;	(*  ~ {LinkedWith:TIID^C6920 (EtherCAT)^ScadaRoom_KouplerUTP (EK1100)^ScadaRoom_KouplerFiber (EK1521)^InletWork_1(EK1501)^InletWork_2 (EK1122)^Term 16 (EK1100)^Term 18 (EL1809)^Channel 7^Input} *)
	STP.PS101B2_Penstock_OpenStat AT %IX13.4 : BOOL;	(*  ~ {LinkedWith:TIID^C6920 (EtherCAT)^ScadaRoom_KouplerUTP (EK1100)^ScadaRoom_KouplerFiber (EK1521)^InletWork_1(EK1501)^InletWork_2 (EK1122)^Term 16 (EK1100)^Term 18 (EL1809)^Channel 8^Input} *)
	STP.PS101B1_Penstock_CloseStat AT %IX13.5 : BOOL;	(*  ~ {LinkedWith:TIID^C6920 (EtherCAT)^ScadaRoom_KouplerUTP (EK1100)^ScadaRoom_KouplerFiber (EK1521)^InletWork_1(EK1501)^InletWork_2 (EK1122)^Term 16 (EK1100)^Term 18 (EL1809)^Channel 9^Input} *)
	STP.PS101B2_Penstock_CloseStat AT %IX13.6 : BOOL;	(*  ~ {LinkedWith:TIID^C6920 (EtherCAT)^ScadaRoom_KouplerUTP (EK1100)^ScadaRoom_KouplerFiber (EK1521)^InletWork_1(EK1501)^InletWork_2 (EK1122)^Term 16 (EK1100)^Term 18 (EL1809)^Channel 10^Input} *)
	STP.XV101B1_SolenoidValveSpray_CloseStat AT %IX13.7 : BOOL;	(*  ~ {LinkedWith:TIID^C6920 (EtherCAT)^ScadaRoom_KouplerUTP (EK1100)^ScadaRoom_KouplerFiber (EK1521)^InletWork_1(EK1501)^InletWork_2 (EK1122)^Term 16 (EK1100)^Term 18 (EL1809)^Channel 11^Input} *)
	STP.XV101B2_SolenoidValveSpray_CloseStat AT %IX14.0 : BOOL;	(*  ~ {LinkedWith:TIID^C6920 (EtherCAT)^ScadaRoom_KouplerUTP (EK1100)^ScadaRoom_KouplerFiber (EK1521)^InletWork_1(EK1501)^InletWork_2 (EK1122)^Term 16 (EK1100)^Term 18 (EL1809)^Channel 12^Input} *)
	STP.XV102B1_ContinuosValveWater_CloseStat AT %IX14.1 : BOOL;	(*  ~ {LinkedWith:TIID^C6920 (EtherCAT)^ScadaRoom_KouplerUTP (EK1100)^ScadaRoom_KouplerFiber (EK1521)^InletWork_1(EK1501)^InletWork_2 (EK1122)^Term 16 (EK1100)^Term 18 (EL1809)^Channel 13^Input} *)
	STP.XV100B1_GritRemovalValve_CloseStat AT %IX14.2 : BOOL;	(*  ~ {LinkedWith:TIID^C6920 (EtherCAT)^ScadaRoom_KouplerUTP (EK1100)^ScadaRoom_KouplerFiber (EK1521)^InletWork_1(EK1501)^InletWork_2 (EK1122)^Term 16 (EK1100)^Term 18 (EL1809)^Channel 14^Input} *)
	STP.XV100B2_GritRemovalValve_CloseStat AT %IX14.3 : BOOL;	(*  ~ {LinkedWith:TIID^C6920 (EtherCAT)^ScadaRoom_KouplerUTP (EK1100)^ScadaRoom_KouplerFiber (EK1521)^InletWork_1(EK1501)^InletWork_2 (EK1122)^Term 16 (EK1100)^Term 18 (EL1809)^Channel 15^Input} *)
	STP.M101B1_EQMixer_OverloadStat AT %IX14.4 : BOOL;	(*  ~ {LinkedWith:TIID^C6920 (EtherCAT)^ScadaRoom_KouplerUTP (EK1100)^ScadaRoom_KouplerFiber (EK1521)^InletWork_1(EK1501)^InletWork_2 (EK1122)^Term 16 (EK1100)^Term 19 (EL1809)^Channel 1^Input} *)
	STP.M101B1_EQMixer_IncompleteStat AT %IX14.5 : BOOL;	(*  ~ {LinkedWith:TIID^C6920 (EtherCAT)^ScadaRoom_KouplerUTP (EK1100)^ScadaRoom_KouplerFiber (EK1521)^InletWork_1(EK1501)^InletWork_2 (EK1122)^Term 16 (EK1100)^Term 19 (EL1809)^Channel 2^Input} *)
	STP.M101B2_EQMixer_OverloadStat AT %IX14.6 : BOOL;	(*  ~ {LinkedWith:TIID^C6920 (EtherCAT)^ScadaRoom_KouplerUTP (EK1100)^ScadaRoom_KouplerFiber (EK1521)^InletWork_1(EK1501)^InletWork_2 (EK1122)^Term 16 (EK1100)^Term 19 (EL1809)^Channel 3^Input} *)
	STP.M101B2_EQMixer_IncompleteStat AT %IX14.7 : BOOL;	(*  ~ {LinkedWith:TIID^C6920 (EtherCAT)^ScadaRoom_KouplerUTP (EK1100)^ScadaRoom_KouplerFiber (EK1521)^InletWork_1(EK1501)^InletWork_2 (EK1122)^Term 16 (EK1100)^Term 19 (EL1809)^Channel 4^Input} *)
	STP.P101B1_EQPump_OverloadStat AT %IX15.0 : BOOL;	(*  ~ {LinkedWith:TIID^C6920 (EtherCAT)^ScadaRoom_KouplerUTP (EK1100)^ScadaRoom_KouplerFiber (EK1521)^InletWork_1(EK1501)^InletWork_2 (EK1122)^Term 16 (EK1100)^Term 19 (EL1809)^Channel 5^Input} *)
	STP.P101B1_EQPump_IncompleteStat AT %IX15.1 : BOOL;	(*  ~ {LinkedWith:TIID^C6920 (EtherCAT)^ScadaRoom_KouplerUTP (EK1100)^ScadaRoom_KouplerFiber (EK1521)^InletWork_1(EK1501)^InletWork_2 (EK1122)^Term 16 (EK1100)^Term 19 (EL1809)^Channel 6^Input} *)
	STP.P101B2_EQPump_OverloadStat AT %IX15.2 : BOOL;	(*  ~ {LinkedWith:TIID^C6920 (EtherCAT)^ScadaRoom_KouplerUTP (EK1100)^ScadaRoom_KouplerFiber (EK1521)^InletWork_1(EK1501)^InletWork_2 (EK1122)^Term 16 (EK1100)^Term 19 (EL1809)^Channel 7^Input} *)
	STP.P101B2_EQPump_IncompleteStat AT %IX15.3 : BOOL;	(*  ~ {LinkedWith:TIID^C6920 (EtherCAT)^ScadaRoom_KouplerUTP (EK1100)^ScadaRoom_KouplerFiber (EK1521)^InletWork_1(EK1501)^InletWork_2 (EK1122)^Term 16 (EK1100)^Term 19 (EL1809)^Channel 8^Input} *)
	STP.PS101B1_Penstock_TripStat AT %IX15.4 : BOOL;	(*  ~ {LinkedWith:TIID^C6920 (EtherCAT)^ScadaRoom_KouplerUTP (EK1100)^ScadaRoom_KouplerFiber (EK1521)^InletWork_1(EK1501)^InletWork_2 (EK1122)^Term 16 (EK1100)^Term 19 (EL1809)^Channel 9^Input} *)
	STP.PSB101B2_Penstock_TripStat AT %IX15.5 : BOOL;	(*  ~ {LinkedWith:TIID^C6920 (EtherCAT)^ScadaRoom_KouplerUTP (EK1100)^ScadaRoom_KouplerFiber (EK1521)^InletWork_1(EK1501)^InletWork_2 (EK1122)^Term 16 (EK1100)^Term 19 (EL1809)^Channel 10^Input} *)
	STP.F101B1_FineScr_OverloadStat AT %IX15.6 : BOOL;	(*  ~ {LinkedWith:TIID^C6920 (EtherCAT)^ScadaRoom_KouplerUTP (EK1100)^ScadaRoom_KouplerFiber (EK1521)^InletWork_1(EK1501)^InletWork_2 (EK1122)^Term 16 (EK1100)^Term 20 (EL1809)^Channel 1^Input} *)
	STP.F101B2_FineScr_OverloadStat AT %IX15.7 : BOOL;	(*  ~ {LinkedWith:TIID^C6920 (EtherCAT)^ScadaRoom_KouplerUTP (EK1100)^ScadaRoom_KouplerFiber (EK1521)^InletWork_1(EK1501)^InletWork_2 (EK1122)^Term 16 (EK1100)^Term 20 (EL1809)^Channel 2^Input} *)
	STP.C102B_ScreeningConveyer_OverloadStat AT %IX16.0 : BOOL;	(*  ~ {LinkedWith:TIID^C6920 (EtherCAT)^ScadaRoom_KouplerUTP (EK1100)^ScadaRoom_KouplerFiber (EK1521)^InletWork_1(EK1501)^InletWork_2 (EK1122)^Term 16 (EK1100)^Term 20 (EL1809)^Channel 3^Input} *)
	STP.C101B_ScreeningCompactor_OverloadStat AT %IX16.1 : BOOL;	(*  ~ {LinkedWith:TIID^C6920 (EtherCAT)^ScadaRoom_KouplerUTP (EK1100)^ScadaRoom_KouplerFiber (EK1521)^InletWork_1(EK1501)^InletWork_2 (EK1122)^Term 16 (EK1100)^Term 20 (EL1809)^Channel 4^Input} *)
	STP.C103B_GritClassifier_OverloadStat AT %IX16.2 : BOOL;	(*  ~ {LinkedWith:TIID^C6920 (EtherCAT)^ScadaRoom_KouplerUTP (EK1100)^ScadaRoom_KouplerFiber (EK1521)^InletWork_1(EK1501)^InletWork_2 (EK1122)^Term 16 (EK1100)^Term 20 (EL1809)^Channel 5^Input} *)
	STP.P102B1_SBRTransferPump_OverloadStat AT %IX16.3 : BOOL;	(*  ~ {LinkedWith:TIID^C6920 (EtherCAT)^ScadaRoom_KouplerUTP (EK1100)^ScadaRoom_KouplerFiber (EK1521)^InletWork_1(EK1501)^InletWork_2 (EK1122)^Term 16 (EK1100)^Term 20 (EL1809)^Channel 6^Input} *)
	STP.P102B1_SBRTransferPump_IncompleteStat AT %IX16.4 : BOOL;	(*  ~ {LinkedWith:TIID^C6920 (EtherCAT)^ScadaRoom_KouplerUTP (EK1100)^ScadaRoom_KouplerFiber (EK1521)^InletWork_1(EK1501)^InletWork_2 (EK1122)^Term 16 (EK1100)^Term 20 (EL1809)^Channel 7^Input} *)
	STP.P102B2_SBRTransferPump_OverloadStat AT %IX16.5 : BOOL;	(*  ~ {LinkedWith:TIID^C6920 (EtherCAT)^ScadaRoom_KouplerUTP (EK1100)^ScadaRoom_KouplerFiber (EK1521)^InletWork_1(EK1501)^InletWork_2 (EK1122)^Term 16 (EK1100)^Term 20 (EL1809)^Channel 8^Input} *)
	STP.P102B2_SBRTransferPump_IncompleteStat AT %IX16.6 : BOOL;	(*  ~ {LinkedWith:TIID^C6920 (EtherCAT)^ScadaRoom_KouplerUTP (EK1100)^ScadaRoom_KouplerFiber (EK1521)^InletWork_1(EK1501)^InletWork_2 (EK1122)^Term 16 (EK1100)^Term 20 (EL1809)^Channel 9^Input} *)
	STP.M101B1_EQMixer_LocalRemoteStat AT %IX16.7 : BOOL;	(*  ~ {LinkedWith:TIID^C6920 (EtherCAT)^ScadaRoom_KouplerUTP (EK1100)^ScadaRoom_KouplerFiber (EK1521)^InletWork_1(EK1501)^InletWork_2 (EK1122)^Term 16 (EK1100)^Term 21 (EL1809)^Channel 1^Input} *)
	STP.M101B2_EQMixer_LocalRemoteStat AT %IX17.0 : BOOL;	(*  ~ {LinkedWith:TIID^C6920 (EtherCAT)^ScadaRoom_KouplerUTP (EK1100)^ScadaRoom_KouplerFiber (EK1521)^InletWork_1(EK1501)^InletWork_2 (EK1122)^Term 16 (EK1100)^Term 21 (EL1809)^Channel 2^Input} *)
	STP.P101B1_EQPump_LocalRemoteStat AT %IX17.1 : BOOL;	(*  ~ {LinkedWith:TIID^C6920 (EtherCAT)^ScadaRoom_KouplerUTP (EK1100)^ScadaRoom_KouplerFiber (EK1521)^InletWork_1(EK1501)^InletWork_2 (EK1122)^Term 16 (EK1100)^Term 21 (EL1809)^Channel 3^Input} *)
	STP.P101B2_EQPump_LocalRemoteStat AT %IX17.2 : BOOL;	(*  ~ {LinkedWith:TIID^C6920 (EtherCAT)^ScadaRoom_KouplerUTP (EK1100)^ScadaRoom_KouplerFiber (EK1521)^InletWork_1(EK1501)^InletWork_2 (EK1122)^Term 16 (EK1100)^Term 21 (EL1809)^Channel 4^Input} *)
	STP.F101B1_FineScr_LocalRemoteStat AT %IX17.3 : BOOL;	(*  ~ {LinkedWith:TIID^C6920 (EtherCAT)^ScadaRoom_KouplerUTP (EK1100)^ScadaRoom_KouplerFiber (EK1521)^InletWork_1(EK1501)^InletWork_2 (EK1122)^Term 16 (EK1100)^Term 21 (EL1809)^Channel 5^Input} *)
	STP.F101B2_FineScr_LocalRemoteStat AT %IX17.4 : BOOL;	(*  ~ {LinkedWith:TIID^C6920 (EtherCAT)^ScadaRoom_KouplerUTP (EK1100)^ScadaRoom_KouplerFiber (EK1521)^InletWork_1(EK1501)^InletWork_2 (EK1122)^Term 16 (EK1100)^Term 21 (EL1809)^Channel 6^Input} *)
	STP.C102B_ScreenConveyer_LocalRemoteStat AT %IX17.5 : BOOL;	(*  ~ {LinkedWith:TIID^C6920 (EtherCAT)^ScadaRoom_KouplerUTP (EK1100)^ScadaRoom_KouplerFiber (EK1521)^InletWork_1(EK1501)^InletWork_2 (EK1122)^Term 16 (EK1100)^Term 21 (EL1809)^Channel 7^Input} *)
	STP.C101B_ScreenCompactor_LocalRemoteStat AT %IX17.6 : BOOL;	(*  ~ {LinkedWith:TIID^C6920 (EtherCAT)^ScadaRoom_KouplerUTP (EK1100)^ScadaRoom_KouplerFiber (EK1521)^InletWork_1(EK1501)^InletWork_2 (EK1122)^Term 16 (EK1100)^Term 21 (EL1809)^Channel 8^Input} *)
	STP.C103BB_GritClasifiier_LocalRemoteStat AT %IX17.7 : BOOL;	(*  ~ {LinkedWith:TIID^C6920 (EtherCAT)^ScadaRoom_KouplerUTP (EK1100)^ScadaRoom_KouplerFiber (EK1521)^InletWork_1(EK1501)^InletWork_2 (EK1122)^Term 16 (EK1100)^Term 21 (EL1809)^Channel 9^Input} *)
	STP.P102B1_SBRTransferPump_LocalRemoteStat AT %IX18.0 : BOOL;	(*  ~ {LinkedWith:TIID^C6920 (EtherCAT)^ScadaRoom_KouplerUTP (EK1100)^ScadaRoom_KouplerFiber (EK1521)^InletWork_1(EK1501)^InletWork_2 (EK1122)^Term 16 (EK1100)^Term 21 (EL1809)^Channel 10^Input} *)
	STP.P102B2_SBRTransferPump_LocalRemoteStat AT %IX18.1 : BOOL;	(*  ~ {LinkedWith:TIID^C6920 (EtherCAT)^ScadaRoom_KouplerUTP (EK1100)^ScadaRoom_KouplerFiber (EK1521)^InletWork_1(EK1501)^InletWork_2 (EK1122)^Term 16 (EK1100)^Term 21 (EL1809)^Channel 11^Input} *)
	STP.PS101B1_Penstock_LocalRemoteStat AT %IX296.2 : BOOL;	(*  ~ {LinkedWith:TIID^C6920 (EtherCAT)^ScadaRoom_KouplerUTP (EK1100)^ScadaRoom_KouplerFiber (EK1521)^InletWork_1(EK1501)^InletWork_2 (EK1122)^Term 16 (EK1100)^Term 21 (EL1809)^Channel 12^Input} *)
	STP.PS101B2_Penstock_LocalRemoteStat AT %IX296.3 : BOOL;	(*  ~ {LinkedWith:TIID^C6920 (EtherCAT)^ScadaRoom_KouplerUTP (EK1100)^ScadaRoom_KouplerFiber (EK1521)^InletWork_1(EK1501)^InletWork_2 (EK1122)^Term 16 (EK1100)^Term 21 (EL1809)^Channel 13^Input} *)
	STP.M101B1_EQMixer_RunStat AT %IX18.2 : BOOL;	(*  ~ {LinkedWith:TIID^C6920 (EtherCAT)^ScadaRoom_KouplerUTP (EK1100)^ScadaRoom_KouplerFiber (EK1521)^InletWork_1(EK1501)^InletWork_2 (EK1122)^Term 16 (EK1100)^Term 22 (EL1809)^Channel 1^Input} *)
	STP.M101B2_EQMixer_RunStat AT %IX18.3 : BOOL;	(*  ~ {LinkedWith:TIID^C6920 (EtherCAT)^ScadaRoom_KouplerUTP (EK1100)^ScadaRoom_KouplerFiber (EK1521)^InletWork_1(EK1501)^InletWork_2 (EK1122)^Term 16 (EK1100)^Term 22 (EL1809)^Channel 2^Input} *)
	STP.P101B1_EQPump_RunStat AT %IX18.4 : BOOL;	(*  ~ {LinkedWith:TIID^C6920 (EtherCAT)^ScadaRoom_KouplerUTP (EK1100)^ScadaRoom_KouplerFiber (EK1521)^InletWork_1(EK1501)^InletWork_2 (EK1122)^Term 16 (EK1100)^Term 22 (EL1809)^Channel 3^Input} *)
	STP.P101B2_EQPump_RunStat AT %IX18.5 : BOOL;	(*  ~ {LinkedWith:TIID^C6920 (EtherCAT)^ScadaRoom_KouplerUTP (EK1100)^ScadaRoom_KouplerFiber (EK1521)^InletWork_1(EK1501)^InletWork_2 (EK1122)^Term 16 (EK1100)^Term 22 (EL1809)^Channel 4^Input} *)
	STP.F101B1_FineScr_RunStat AT %IX18.6 : BOOL;	(*  ~ {LinkedWith:TIID^C6920 (EtherCAT)^ScadaRoom_KouplerUTP (EK1100)^ScadaRoom_KouplerFiber (EK1521)^InletWork_1(EK1501)^InletWork_2 (EK1122)^Term 16 (EK1100)^Term 22 (EL1809)^Channel 5^Input} *)
	STP.F101B2_FineScr_RunStat AT %IX18.7 : BOOL;	(*  ~ {LinkedWith:TIID^C6920 (EtherCAT)^ScadaRoom_KouplerUTP (EK1100)^ScadaRoom_KouplerFiber (EK1521)^InletWork_1(EK1501)^InletWork_2 (EK1122)^Term 16 (EK1100)^Term 22 (EL1809)^Channel 6^Input} *)
	STP.C102B_ScreenConveyer_RunStat AT %IX19.0 : BOOL;	(*  ~ {LinkedWith:TIID^C6920 (EtherCAT)^ScadaRoom_KouplerUTP (EK1100)^ScadaRoom_KouplerFiber (EK1521)^InletWork_1(EK1501)^InletWork_2 (EK1122)^Term 16 (EK1100)^Term 22 (EL1809)^Channel 7^Input} *)
	STP.C101B_ScreenCompactor_RunStat AT %IX19.1 : BOOL;	(*  ~ {LinkedWith:TIID^C6920 (EtherCAT)^ScadaRoom_KouplerUTP (EK1100)^ScadaRoom_KouplerFiber (EK1521)^InletWork_1(EK1501)^InletWork_2 (EK1122)^Term 16 (EK1100)^Term 22 (EL1809)^Channel 8^Input} *)
	STP.C103B_GritClasifier_RunStat AT %IX19.2 : BOOL;	(*  ~ {LinkedWith:TIID^C6920 (EtherCAT)^ScadaRoom_KouplerUTP (EK1100)^ScadaRoom_KouplerFiber (EK1521)^InletWork_1(EK1501)^InletWork_2 (EK1122)^Term 16 (EK1100)^Term 22 (EL1809)^Channel 9^Input} *)
	STP.P102B1_SBRTransferPump_RunStat AT %IX19.3 : BOOL;	(*  ~ {LinkedWith:TIID^C6920 (EtherCAT)^ScadaRoom_KouplerUTP (EK1100)^ScadaRoom_KouplerFiber (EK1521)^InletWork_1(EK1501)^InletWork_2 (EK1122)^Term 16 (EK1100)^Term 22 (EL1809)^Channel 10^Input} *)
	STP.P102B2_SBRTransferPump_RunStat AT %IX19.4 : BOOL;	(*  ~ {LinkedWith:TIID^C6920 (EtherCAT)^ScadaRoom_KouplerUTP (EK1100)^ScadaRoom_KouplerFiber (EK1521)^InletWork_1(EK1501)^InletWork_2 (EK1122)^Term 16 (EK1100)^Term 22 (EL1809)^Channel 11^Input} *)
	STP.M101B1_EQMixer_EStopStat AT %IX19.5 : BOOL;	(*  ~ {LinkedWith:TIID^C6920 (EtherCAT)^ScadaRoom_KouplerUTP (EK1100)^ScadaRoom_KouplerFiber (EK1521)^InletWork_1(EK1501)^InletWork_2 (EK1122)^Term 16 (EK1100)^Term 23 (EL1809)^Channel 1^Input} *)
	STP.M101B2_EQMixer_EStopStat AT %IX19.6 : BOOL;	(*  ~ {LinkedWith:TIID^C6920 (EtherCAT)^ScadaRoom_KouplerUTP (EK1100)^ScadaRoom_KouplerFiber (EK1521)^InletWork_1(EK1501)^InletWork_2 (EK1122)^Term 16 (EK1100)^Term 23 (EL1809)^Channel 2^Input} *)
	STP.P101B1_EQPump_EStopStat AT %IX19.7 : BOOL;	(*  ~ {LinkedWith:TIID^C6920 (EtherCAT)^ScadaRoom_KouplerUTP (EK1100)^ScadaRoom_KouplerFiber (EK1521)^InletWork_1(EK1501)^InletWork_2 (EK1122)^Term 16 (EK1100)^Term 23 (EL1809)^Channel 3^Input} *)
	STP.P101B2_EQPump_EStopStat AT %IX20.0 : BOOL;	(*  ~ {LinkedWith:TIID^C6920 (EtherCAT)^ScadaRoom_KouplerUTP (EK1100)^ScadaRoom_KouplerFiber (EK1521)^InletWork_1(EK1501)^InletWork_2 (EK1122)^Term 16 (EK1100)^Term 23 (EL1809)^Channel 4^Input} *)
	STP.F101B1_FineScr_EStopStat AT %IX20.1 : BOOL;	(*  ~ {LinkedWith:TIID^C6920 (EtherCAT)^ScadaRoom_KouplerUTP (EK1100)^ScadaRoom_KouplerFiber (EK1521)^InletWork_1(EK1501)^InletWork_2 (EK1122)^Term 16 (EK1100)^Term 23 (EL1809)^Channel 5^Input} *)
	STP.F101B2_FineScr_EStopStat AT %IX20.2 : BOOL;	(*  ~ {LinkedWith:TIID^C6920 (EtherCAT)^ScadaRoom_KouplerUTP (EK1100)^ScadaRoom_KouplerFiber (EK1521)^InletWork_1(EK1501)^InletWork_2 (EK1122)^Term 16 (EK1100)^Term 23 (EL1809)^Channel 6^Input} *)
	STP.C102B_ScreenConveyer_EStopStat AT %IX20.3 : BOOL;	(*  ~ {LinkedWith:TIID^C6920 (EtherCAT)^ScadaRoom_KouplerUTP (EK1100)^ScadaRoom_KouplerFiber (EK1521)^InletWork_1(EK1501)^InletWork_2 (EK1122)^Term 16 (EK1100)^Term 23 (EL1809)^Channel 7^Input} *)
	STP.C101B_ScreenCompactor_EStopStat AT %IX20.4 : BOOL;	(*  ~ {LinkedWith:TIID^C6920 (EtherCAT)^ScadaRoom_KouplerUTP (EK1100)^ScadaRoom_KouplerFiber (EK1521)^InletWork_1(EK1501)^InletWork_2 (EK1122)^Term 16 (EK1100)^Term 23 (EL1809)^Channel 8^Input} *)
	STP.C103B_GritClasifier_EStopStat AT %IX20.5 : BOOL;	(*  ~ {LinkedWith:TIID^C6920 (EtherCAT)^ScadaRoom_KouplerUTP (EK1100)^ScadaRoom_KouplerFiber (EK1521)^InletWork_1(EK1501)^InletWork_2 (EK1122)^Term 16 (EK1100)^Term 23 (EL1809)^Channel 9^Input} *)
	STP.P102B1_SBRTransferPump_EStopStat AT %IX20.6 : BOOL;	(*  ~ {LinkedWith:TIID^C6920 (EtherCAT)^ScadaRoom_KouplerUTP (EK1100)^ScadaRoom_KouplerFiber (EK1521)^InletWork_1(EK1501)^InletWork_2 (EK1122)^Term 16 (EK1100)^Term 23 (EL1809)^Channel 10^Input} *)
	STP.P102B2_SBRTransferPump_EStopStat AT %IX20.7 : BOOL;	(*  ~ {LinkedWith:TIID^C6920 (EtherCAT)^ScadaRoom_KouplerUTP (EK1100)^ScadaRoom_KouplerFiber (EK1521)^InletWork_1(EK1501)^InletWork_2 (EK1122)^Term 16 (EK1100)^Term 23 (EL1809)^Channel 11^Input} *)
	STP.VE801A_SuctionFan_OnOffStat AT %IX21.0 : BOOL;	(*  ~ {LinkedWith:TIID^C6920 (EtherCAT)^ScadaRoom_KouplerUTP (EK1100)^ScadaRoom_KouplerFiber (EK1521)^InletWork_1(EK1501)^InletWork_2 (EK1122)^Term 16 (EK1100)^Term 24 (EL1809)^Channel 1^Input} *)
	STP.P802A_CirculationPump_OnOffStat AT %IX21.1 : BOOL;	(*  ~ {LinkedWith:TIID^C6920 (EtherCAT)^ScadaRoom_KouplerUTP (EK1100)^ScadaRoom_KouplerFiber (EK1521)^InletWork_1(EK1501)^InletWork_2 (EK1122)^Term 16 (EK1100)^Term 24 (EL1809)^Channel 2^Input} *)
	STP.P803A_CirculationPump_OnOffStat AT %IX21.2 : BOOL;	(*  ~ {LinkedWith:TIID^C6920 (EtherCAT)^ScadaRoom_KouplerUTP (EK1100)^ScadaRoom_KouplerFiber (EK1521)^InletWork_1(EK1501)^InletWork_2 (EK1122)^Term 16 (EK1100)^Term 24 (EL1809)^Channel 3^Input} *)
	STP.P804A_CirculationPump_OnOffStat AT %IX21.3 : BOOL;	(*  ~ {LinkedWith:TIID^C6920 (EtherCAT)^ScadaRoom_KouplerUTP (EK1100)^ScadaRoom_KouplerFiber (EK1521)^InletWork_1(EK1501)^InletWork_2 (EK1122)^Term 16 (EK1100)^Term 24 (EL1809)^Channel 4^Input} *)
	STP.P805A1_H2S04Pump_OnOffStat AT %IX21.4 : BOOL;	(*  ~ {LinkedWith:TIID^C6920 (EtherCAT)^ScadaRoom_KouplerUTP (EK1100)^ScadaRoom_KouplerFiber (EK1521)^InletWork_1(EK1501)^InletWork_2 (EK1122)^Term 16 (EK1100)^Term 24 (EL1809)^Channel 5^Input} *)
	STP.P805A2_H2S04Pump_OnOffStat AT %IX21.5 : BOOL;	(*  ~ {LinkedWith:TIID^C6920 (EtherCAT)^ScadaRoom_KouplerUTP (EK1100)^ScadaRoom_KouplerFiber (EK1521)^InletWork_1(EK1501)^InletWork_2 (EK1122)^Term 16 (EK1100)^Term 24 (EL1809)^Channel 6^Input} *)
	STP.P806A1_NAOHPump_OnOffStat AT %IX21.6 : BOOL;	(*  ~ {LinkedWith:TIID^C6920 (EtherCAT)^ScadaRoom_KouplerUTP (EK1100)^ScadaRoom_KouplerFiber (EK1521)^InletWork_1(EK1501)^InletWork_2 (EK1122)^Term 16 (EK1100)^Term 24 (EL1809)^Channel 7^Input} *)
	STP.P806A2_NAOHPump_OnOffStat AT %IX21.7 : BOOL;	(*  ~ {LinkedWith:TIID^C6920 (EtherCAT)^ScadaRoom_KouplerUTP (EK1100)^ScadaRoom_KouplerFiber (EK1521)^InletWork_1(EK1501)^InletWork_2 (EK1122)^Term 16 (EK1100)^Term 24 (EL1809)^Channel 8^Input} *)
	STP.P807A1_NAOCLPump_OnOffStat AT %IX22.0 : BOOL;	(*  ~ {LinkedWith:TIID^C6920 (EtherCAT)^ScadaRoom_KouplerUTP (EK1100)^ScadaRoom_KouplerFiber (EK1521)^InletWork_1(EK1501)^InletWork_2 (EK1122)^Term 16 (EK1100)^Term 24 (EL1809)^Channel 9^Input} *)
	STP.P807A2_NAOCLPump_OnOffStat AT %IX22.1 : BOOL;	(*  ~ {LinkedWith:TIID^C6920 (EtherCAT)^ScadaRoom_KouplerUTP (EK1100)^ScadaRoom_KouplerFiber (EK1521)^InletWork_1(EK1501)^InletWork_2 (EK1122)^Term 16 (EK1100)^Term 24 (EL1809)^Channel 10^Input} *)
	STP.VE801A_SuctionFan_OverloadStat AT %IX22.2 : BOOL;	(*  ~ {LinkedWith:TIID^C6920 (EtherCAT)^ScadaRoom_KouplerUTP (EK1100)^ScadaRoom_KouplerFiber (EK1521)^InletWork_1(EK1501)^InletWork_2 (EK1122)^Term 16 (EK1100)^Term 24 (EL1809)^Channel 11^Input} *)
	STP.P802A_CirculationPump_OverloadStat AT %IX22.3 : BOOL;	(*  ~ {LinkedWith:TIID^C6920 (EtherCAT)^ScadaRoom_KouplerUTP (EK1100)^ScadaRoom_KouplerFiber (EK1521)^InletWork_1(EK1501)^InletWork_2 (EK1122)^Term 16 (EK1100)^Term 24 (EL1809)^Channel 12^Input} *)
	STP.P803A_CirculationPump_OverloadStat AT %IX22.4 : BOOL;	(*  ~ {LinkedWith:TIID^C6920 (EtherCAT)^ScadaRoom_KouplerUTP (EK1100)^ScadaRoom_KouplerFiber (EK1521)^InletWork_1(EK1501)^InletWork_2 (EK1122)^Term 16 (EK1100)^Term 24 (EL1809)^Channel 13^Input} *)
	STP.P804A_CirculationPump_OverloadStat AT %IX22.5 : BOOL;	(*  ~ {LinkedWith:TIID^C6920 (EtherCAT)^ScadaRoom_KouplerUTP (EK1100)^ScadaRoom_KouplerFiber (EK1521)^InletWork_1(EK1501)^InletWork_2 (EK1122)^Term 16 (EK1100)^Term 24 (EL1809)^Channel 14^Input} *)
	STP.P805A1_H2S04Pump_OverloadStat AT %IX22.6 : BOOL;	(*  ~ {LinkedWith:TIID^C6920 (EtherCAT)^ScadaRoom_KouplerUTP (EK1100)^ScadaRoom_KouplerFiber (EK1521)^InletWork_1(EK1501)^InletWork_2 (EK1122)^Term 16 (EK1100)^Term 24 (EL1809)^Channel 15^Input} *)
	STP.P805A2_H2S04Pump_OverloadStat AT %IX22.7 : BOOL;	(*  ~ {LinkedWith:TIID^C6920 (EtherCAT)^ScadaRoom_KouplerUTP (EK1100)^ScadaRoom_KouplerFiber (EK1521)^InletWork_1(EK1501)^InletWork_2 (EK1122)^Term 16 (EK1100)^Term 24 (EL1809)^Channel 16^Input} *)
	STP.P806A1_NAOHPump_OverloadStat AT %IX23.0 : BOOL;	(*  ~ {LinkedWith:TIID^C6920 (EtherCAT)^ScadaRoom_KouplerUTP (EK1100)^ScadaRoom_KouplerFiber (EK1521)^InletWork_1(EK1501)^InletWork_2 (EK1122)^Term 16 (EK1100)^Term 25 (EL1809)^Channel 1^Input} *)
	STP.P806A2_NAOHPump_OverloadStat AT %IX23.1 : BOOL;	(*  ~ {LinkedWith:TIID^C6920 (EtherCAT)^ScadaRoom_KouplerUTP (EK1100)^ScadaRoom_KouplerFiber (EK1521)^InletWork_1(EK1501)^InletWork_2 (EK1122)^Term 16 (EK1100)^Term 25 (EL1809)^Channel 2^Input} *)
	STP.P807A1_NAOCLPump_OverloadStat AT %IX23.2 : BOOL;	(*  ~ {LinkedWith:TIID^C6920 (EtherCAT)^ScadaRoom_KouplerUTP (EK1100)^ScadaRoom_KouplerFiber (EK1521)^InletWork_1(EK1501)^InletWork_2 (EK1122)^Term 16 (EK1100)^Term 25 (EL1809)^Channel 3^Input} *)
	STP.P807A2_NAOCLPump_OverloadStat AT %IX23.3 : BOOL;	(*  ~ {LinkedWith:TIID^C6920 (EtherCAT)^ScadaRoom_KouplerUTP (EK1100)^ScadaRoom_KouplerFiber (EK1521)^InletWork_1(EK1501)^InletWork_2 (EK1122)^Term 16 (EK1100)^Term 25 (EL1809)^Channel 4^Input} *)
	STP.VE801A_SuctionFan_EStopStat AT %IX23.4 : BOOL;	(*  ~ {LinkedWith:TIID^C6920 (EtherCAT)^ScadaRoom_KouplerUTP (EK1100)^ScadaRoom_KouplerFiber (EK1521)^InletWork_1(EK1501)^InletWork_2 (EK1122)^Term 16 (EK1100)^Term 25 (EL1809)^Channel 5^Input} *)
	STP.P802A_CirculationPump_EStopStat AT %IX23.5 : BOOL;	(*  ~ {LinkedWith:TIID^C6920 (EtherCAT)^ScadaRoom_KouplerUTP (EK1100)^ScadaRoom_KouplerFiber (EK1521)^InletWork_1(EK1501)^InletWork_2 (EK1122)^Term 16 (EK1100)^Term 25 (EL1809)^Channel 6^Input} *)
	STP.P803A_CirculationPump_EStopStat AT %IX23.6 : BOOL;	(*  ~ {LinkedWith:TIID^C6920 (EtherCAT)^ScadaRoom_KouplerUTP (EK1100)^ScadaRoom_KouplerFiber (EK1521)^InletWork_1(EK1501)^InletWork_2 (EK1122)^Term 16 (EK1100)^Term 25 (EL1809)^Channel 7^Input} *)
	STP.P804A_CirculationPump_EStopStat AT %IX23.7 : BOOL;	(*  ~ {LinkedWith:TIID^C6920 (EtherCAT)^ScadaRoom_KouplerUTP (EK1100)^ScadaRoom_KouplerFiber (EK1521)^InletWork_1(EK1501)^InletWork_2 (EK1122)^Term 16 (EK1100)^Term 25 (EL1809)^Channel 8^Input} *)
	STP.P805A1_H2S04Pump_EStopStat AT %IX24.0 : BOOL;	(*  ~ {LinkedWith:TIID^C6920 (EtherCAT)^ScadaRoom_KouplerUTP (EK1100)^ScadaRoom_KouplerFiber (EK1521)^InletWork_1(EK1501)^InletWork_2 (EK1122)^Term 16 (EK1100)^Term 25 (EL1809)^Channel 9^Input} *)
	STP.P805A2_H2S04Pump_EStopStat AT %IX24.1 : BOOL;	(*  ~ {LinkedWith:TIID^C6920 (EtherCAT)^ScadaRoom_KouplerUTP (EK1100)^ScadaRoom_KouplerFiber (EK1521)^InletWork_1(EK1501)^InletWork_2 (EK1122)^Term 16 (EK1100)^Term 25 (EL1809)^Channel 10^Input} *)
	STP.P806A1_NAOHPump_EStopStat AT %IX24.2 : BOOL;	(*  ~ {LinkedWith:TIID^C6920 (EtherCAT)^ScadaRoom_KouplerUTP (EK1100)^ScadaRoom_KouplerFiber (EK1521)^InletWork_1(EK1501)^InletWork_2 (EK1122)^Term 16 (EK1100)^Term 25 (EL1809)^Channel 11^Input} *)
	STP.P806A2_NAOHPump_EStopStat AT %IX24.3 : BOOL;	(*  ~ {LinkedWith:TIID^C6920 (EtherCAT)^ScadaRoom_KouplerUTP (EK1100)^ScadaRoom_KouplerFiber (EK1521)^InletWork_1(EK1501)^InletWork_2 (EK1122)^Term 16 (EK1100)^Term 25 (EL1809)^Channel 12^Input} *)
	STP.P807A1_NAOCLPump_EStopStat AT %IX24.4 : BOOL;	(*  ~ {LinkedWith:TIID^C6920 (EtherCAT)^ScadaRoom_KouplerUTP (EK1100)^ScadaRoom_KouplerFiber (EK1521)^InletWork_1(EK1501)^InletWork_2 (EK1122)^Term 16 (EK1100)^Term 25 (EL1809)^Channel 13^Input} *)
	STP.P807A2_NAOCLPump_EStopStat AT %IX24.5 : BOOL;	(*  ~ {LinkedWith:TIID^C6920 (EtherCAT)^ScadaRoom_KouplerUTP (EK1100)^ScadaRoom_KouplerFiber (EK1521)^InletWork_1(EK1501)^InletWork_2 (EK1122)^Term 16 (EK1100)^Term 25 (EL1809)^Channel 14^Input} *)
	STP.XV101B1_SolenoidValveSpray_OpenCmd AT %QX80.0 : BOOL;	(*  ~ {LinkedWith:TIID^C6920 (EtherCAT)^ScadaRoom_KouplerUTP (EK1100)^ScadaRoom_KouplerFiber (EK1521)^InletWork_1(EK1501)^InletWork_2 (EK1122)^Term 16 (EK1100)^Term 26 (EL2809)^Channel 1^Output} *)
	STP.XV101B2_SolenoidValveSpray_OpenCmd AT %QX8.1 : BOOL;	(*  ~ {LinkedWith:TIID^C6920 (EtherCAT)^ScadaRoom_KouplerUTP (EK1100)^ScadaRoom_KouplerFiber (EK1521)^InletWork_1(EK1501)^InletWork_2 (EK1122)^Term 16 (EK1100)^Term 26 (EL2809)^Channel 2^Output} *)
	STP.XV102B1_ContinuosValveWater_OpenCmd AT %QX8.2 : BOOL;	(*  ~ {LinkedWith:TIID^C6920 (EtherCAT)^ScadaRoom_KouplerUTP (EK1100)^ScadaRoom_KouplerFiber (EK1521)^InletWork_1(EK1501)^InletWork_2 (EK1122)^Term 16 (EK1100)^Term 26 (EL2809)^Channel 3^Output} *)
	STP.F101B1_FineScr_RunCmd AT %QX4.4 : BOOL;	(*  ~ {LinkedWith:TIID^C6920 (EtherCAT)^ScadaRoom_KouplerUTP (EK1100)^ScadaRoom_KouplerFiber (EK1521)^InletWork_1(EK1501)^InletWork_2 (EK1122)^Term 16 (EK1100)^Term 26 (EL2809)^Channel 5^Output} *)
	STP.F101B2_FineScr_RunCmd AT %QX4.5 : BOOL;	(*  ~ {LinkedWith:TIID^C6920 (EtherCAT)^ScadaRoom_KouplerUTP (EK1100)^ScadaRoom_KouplerFiber (EK1521)^InletWork_1(EK1501)^InletWork_2 (EK1122)^Term 16 (EK1100)^Term 26 (EL2809)^Channel 6^Output} *)
	STP.C102B_ScreenConveyer_RunCmd AT %QX4.6 : BOOL;	(*  ~ {LinkedWith:TIID^C6920 (EtherCAT)^ScadaRoom_KouplerUTP (EK1100)^ScadaRoom_KouplerFiber (EK1521)^InletWork_1(EK1501)^InletWork_2 (EK1122)^Term 16 (EK1100)^Term 26 (EL2809)^Channel 7^Output} *)
	STP.C101B_ScreenCompactor_RunCmd AT %QX4.7 : BOOL;	(*  ~ {LinkedWith:TIID^C6920 (EtherCAT)^ScadaRoom_KouplerUTP (EK1100)^ScadaRoom_KouplerFiber (EK1521)^InletWork_1(EK1501)^InletWork_2 (EK1122)^Term 16 (EK1100)^Term 26 (EL2809)^Channel 8^Output} *)
	STP.C103B_GritClasifier_RunCmd AT %QX5.0 : BOOL;	(*  ~ {LinkedWith:TIID^C6920 (EtherCAT)^ScadaRoom_KouplerUTP (EK1100)^ScadaRoom_KouplerFiber (EK1521)^InletWork_1(EK1501)^InletWork_2 (EK1122)^Term 16 (EK1100)^Term 26 (EL2809)^Channel 9^Output} *)
	STP.PS101B1_Penstock_OpenCmd AT %QX5.1 : BOOL;	(*  ~ {LinkedWith:TIID^C6920 (EtherCAT)^ScadaRoom_KouplerUTP (EK1100)^ScadaRoom_KouplerFiber (EK1521)^InletWork_1(EK1501)^InletWork_2 (EK1122)^Term 16 (EK1100)^Term 26 (EL2809)^Channel 10^Output} *)
	STP.PS101B1_Penstock_CloseCmd AT %QX5.2 : BOOL;	(*  ~ {LinkedWith:TIID^C6920 (EtherCAT)^ScadaRoom_KouplerUTP (EK1100)^ScadaRoom_KouplerFiber (EK1521)^InletWork_1(EK1501)^InletWork_2 (EK1122)^Term 16 (EK1100)^Term 26 (EL2809)^Channel 11^Output} *)
	STP.PS101B2_Penstock_OpenCmd AT %QX5.3 : BOOL;	(*  ~ {LinkedWith:TIID^C6920 (EtherCAT)^ScadaRoom_KouplerUTP (EK1100)^ScadaRoom_KouplerFiber (EK1521)^InletWork_1(EK1501)^InletWork_2 (EK1122)^Term 16 (EK1100)^Term 26 (EL2809)^Channel 12^Output} *)
	STP.PS101B2_Penstock_CloseCmd AT %QX5.4 : BOOL;	(*  ~ {LinkedWith:TIID^C6920 (EtherCAT)^ScadaRoom_KouplerUTP (EK1100)^ScadaRoom_KouplerFiber (EK1521)^InletWork_1(EK1501)^InletWork_2 (EK1122)^Term 16 (EK1100)^Term 26 (EL2809)^Channel 13^Output} *)
	STP.XV100B1_GritRemovalValve_OpenCmd AT %QX5.5 : BOOL;	(*  ~ {LinkedWith:TIID^C6920 (EtherCAT)^ScadaRoom_KouplerUTP (EK1100)^ScadaRoom_KouplerFiber (EK1521)^InletWork_1(EK1501)^InletWork_2 (EK1122)^Term 16 (EK1100)^Term 26 (EL2809)^Channel 14^Output} *)
	STP.XV100B2_GritRemovalValve_OpenCmd AT %QX5.6 : BOOL;	(*  ~ {LinkedWith:TIID^C6920 (EtherCAT)^ScadaRoom_KouplerUTP (EK1100)^ScadaRoom_KouplerFiber (EK1521)^InletWork_1(EK1501)^InletWork_2 (EK1122)^Term 16 (EK1100)^Term 26 (EL2809)^Channel 15^Output} *)
	STP.P101B1_EQPump_RunCmd AT %QX5.7 : BOOL;	(*  ~ {LinkedWith:TIID^C6920 (EtherCAT)^ScadaRoom_KouplerUTP (EK1100)^ScadaRoom_KouplerFiber (EK1521)^InletWork_1(EK1501)^InletWork_2 (EK1122)^Term 16 (EK1100)^Term 27 (EL2809)^Channel 1^Output} *)
	STP.P101B2_EQPump_RunCmd AT %QX6.0 : BOOL;	(*  ~ {LinkedWith:TIID^C6920 (EtherCAT)^ScadaRoom_KouplerUTP (EK1100)^ScadaRoom_KouplerFiber (EK1521)^InletWork_1(EK1501)^InletWork_2 (EK1122)^Term 16 (EK1100)^Term 27 (EL2809)^Channel 2^Output} *)
	STP.M101B1_EQMixer_RunCmd AT %QX6.1 : BOOL;	(*  ~ {LinkedWith:TIID^C6920 (EtherCAT)^ScadaRoom_KouplerUTP (EK1100)^ScadaRoom_KouplerFiber (EK1521)^InletWork_1(EK1501)^InletWork_2 (EK1122)^Term 16 (EK1100)^Term 27 (EL2809)^Channel 3^Output} *)
	STP.M101B2_EQMixer_RunCmd AT %QX6.2 : BOOL;	(*  ~ {LinkedWith:TIID^C6920 (EtherCAT)^ScadaRoom_KouplerUTP (EK1100)^ScadaRoom_KouplerFiber (EK1521)^InletWork_1(EK1501)^InletWork_2 (EK1122)^Term 16 (EK1100)^Term 27 (EL2809)^Channel 4^Output} *)
	STP.P102B1_SBRTransferPump_RunCmd AT %QX6.3 : BOOL;	(*  ~ {LinkedWith:TIID^C6920 (EtherCAT)^ScadaRoom_KouplerUTP (EK1100)^ScadaRoom_KouplerFiber (EK1521)^InletWork_1(EK1501)^InletWork_2 (EK1122)^Term 16 (EK1100)^Term 27 (EL2809)^Channel 5^Output} *)
	STP.P102B2_SBRTransferPump_RunCmd AT %QX6.4 : BOOL;	(*  ~ {LinkedWith:TIID^C6920 (EtherCAT)^ScadaRoom_KouplerUTP (EK1100)^ScadaRoom_KouplerFiber (EK1521)^InletWork_1(EK1501)^InletWork_2 (EK1122)^Term 16 (EK1100)^Term 27 (EL2809)^Channel 6^Output} *)
	STP.AUX101B_EQFloatSensor_AlarmS2 AT %QX6.5 : BOOL;	(*  ~ {LinkedWith:TIID^C6920 (EtherCAT)^ScadaRoom_KouplerUTP (EK1100)^ScadaRoom_KouplerFiber (EK1521)^InletWork_1(EK1501)^InletWork_2 (EK1122)^Term 16 (EK1100)^Term 27 (EL2809)^Channel 7^Output} *)
	STP.AUX104B_SBRFloatSensor_AlarmS2 AT %QX6.6 : BOOL;	(*  ~ {LinkedWith:TIID^C6920 (EtherCAT)^ScadaRoom_KouplerUTP (EK1100)^ScadaRoom_KouplerFiber (EK1521)^InletWork_1(EK1501)^InletWork_2 (EK1122)^Term 16 (EK1100)^Term 27 (EL2809)^Channel 8^Output} *)
	STP.AUX105B_StreamSensorOverflow_AlarmS2 AT %QX6.7 : BOOL;	(*  ~ {LinkedWith:TIID^C6920 (EtherCAT)^ScadaRoom_KouplerUTP (EK1100)^ScadaRoom_KouplerFiber (EK1521)^InletWork_1(EK1501)^InletWork_2 (EK1122)^Term 16 (EK1100)^Term 27 (EL2809)^Channel 9^Output} *)
	STP.TMT02_FanStatus AT %IX36.0 : BOOL;	(*  ~ {LinkedWith:TIID^C6920 (EtherCAT)^ScadaRoom_KouplerUTP (EK1100)^ScadaRoom_KouplerFiber (EK1521)^BlowerHouse_2 (EK1501)^Term 29 (EL1809)^Channel 1^Input} *)
	STP.DP02_DoorPanelStatus AT %IX36.1 : BOOL;	(*  ~ {LinkedWith:TIID^C6920 (EtherCAT)^ScadaRoom_KouplerUTP (EK1100)^ScadaRoom_KouplerFiber (EK1521)^BlowerHouse_2 (EK1501)^Term 29 (EL1809)^Channel 2^Input} *)
	STP.XV261A_DecanterR1_OverloadStat AT %IX36.2 : BOOL;	(*  ~ {LinkedWith:TIID^C6920 (EtherCAT)^ScadaRoom_KouplerUTP (EK1100)^ScadaRoom_KouplerFiber (EK1521)^BlowerHouse_2 (EK1501)^BlowerHouse_1 (EK1122)^Term 42 (EK1100)^Term 43 (EL1809)^Channel 3^Input} *)
	STP.XV262A_DecanterR2_OverloadStat AT %IX36.3 : BOOL;	(*  ~ {LinkedWith:TIID^C6920 (EtherCAT)^ScadaRoom_KouplerUTP (EK1100)^ScadaRoom_KouplerFiber (EK1521)^BlowerHouse_2 (EK1501)^BlowerHouse_1 (EK1122)^Term 42 (EK1100)^Term 43 (EL1809)^Channel 4^Input} *)
	STP.XV263A_DecanterR3_OverloadStat AT %IX36.4 : BOOL;	(*  ~ {LinkedWith:TIID^C6920 (EtherCAT)^ScadaRoom_KouplerUTP (EK1100)^ScadaRoom_KouplerFiber (EK1521)^BlowerHouse_2 (EK1501)^BlowerHouse_1 (EK1122)^Term 42 (EK1100)^Term 43 (EL1809)^Channel 5^Input} *)
	STP.XV264A_DecanterR4_OverloadStat AT %IX36.5 : BOOL;	(*  ~ {LinkedWith:TIID^C6920 (EtherCAT)^ScadaRoom_KouplerUTP (EK1100)^ScadaRoom_KouplerFiber (EK1521)^BlowerHouse_2 (EK1501)^BlowerHouse_1 (EK1122)^Term 42 (EK1100)^Term 43 (EL1809)^Channel 6^Input} *)
	STP.M200A1A_MixerR1_RunStat AT %IX36.6 : BOOL;	(*  ~ {LinkedWith:TIID^C6920 (EtherCAT)^ScadaRoom_KouplerUTP (EK1100)^ScadaRoom_KouplerFiber (EK1521)^BlowerHouse_2 (EK1501)^BlowerHouse_1 (EK1122)^Term 42 (EK1100)^Term 44 (EL1809)^Channel 1^Input} *)
	STP.M200A1B_MixerR1_RunStat AT %IX36.7 : BOOL;	(*  ~ {LinkedWith:TIID^C6920 (EtherCAT)^ScadaRoom_KouplerUTP (EK1100)^ScadaRoom_KouplerFiber (EK1521)^BlowerHouse_2 (EK1501)^BlowerHouse_1 (EK1122)^Term 42 (EK1100)^Term 44 (EL1809)^Channel 2^Input} *)
	STP.M200A1C_MixerR1_RunStat AT %IX37.0 : BOOL;	(*  ~ {LinkedWith:TIID^C6920 (EtherCAT)^ScadaRoom_KouplerUTP (EK1100)^ScadaRoom_KouplerFiber (EK1521)^BlowerHouse_2 (EK1501)^BlowerHouse_1 (EK1122)^Term 42 (EK1100)^Term 44 (EL1809)^Channel 3^Input} *)
	STP.M200A2A_MixerR2_RunStat AT %IX37.1 : BOOL;	(*  ~ {LinkedWith:TIID^C6920 (EtherCAT)^ScadaRoom_KouplerUTP (EK1100)^ScadaRoom_KouplerFiber (EK1521)^BlowerHouse_2 (EK1501)^BlowerHouse_1 (EK1122)^Term 42 (EK1100)^Term 44 (EL1809)^Channel 4^Input} *)
	STP.M200A2B_MixerR2_RunStat AT %IX37.2 : BOOL;	(*  ~ {LinkedWith:TIID^C6920 (EtherCAT)^ScadaRoom_KouplerUTP (EK1100)^ScadaRoom_KouplerFiber (EK1521)^BlowerHouse_2 (EK1501)^BlowerHouse_1 (EK1122)^Term 42 (EK1100)^Term 44 (EL1809)^Channel 5^Input} *)
	STP.M200A2C_MixerR2_RunStat AT %IX37.3 : BOOL;	(*  ~ {LinkedWith:TIID^C6920 (EtherCAT)^ScadaRoom_KouplerUTP (EK1100)^ScadaRoom_KouplerFiber (EK1521)^BlowerHouse_2 (EK1501)^BlowerHouse_1 (EK1122)^Term 42 (EK1100)^Term 44 (EL1809)^Channel 6^Input} *)
	STP.M200A3A_MixerR3_RunStat AT %IX37.4 : BOOL;	(*  ~ {LinkedWith:TIID^C6920 (EtherCAT)^ScadaRoom_KouplerUTP (EK1100)^ScadaRoom_KouplerFiber (EK1521)^BlowerHouse_2 (EK1501)^BlowerHouse_1 (EK1122)^Term 42 (EK1100)^Term 44 (EL1809)^Channel 7^Input} *)
	STP.M200A3B_MixerR3_RunStat AT %IX37.5 : BOOL;	(*  ~ {LinkedWith:TIID^C6920 (EtherCAT)^ScadaRoom_KouplerUTP (EK1100)^ScadaRoom_KouplerFiber (EK1521)^BlowerHouse_2 (EK1501)^BlowerHouse_1 (EK1122)^Term 42 (EK1100)^Term 44 (EL1809)^Channel 8^Input} *)
	STP.M200A3C_MixerR3_RunStat AT %IX37.6 : BOOL;	(*  ~ {LinkedWith:TIID^C6920 (EtherCAT)^ScadaRoom_KouplerUTP (EK1100)^ScadaRoom_KouplerFiber (EK1521)^BlowerHouse_2 (EK1501)^BlowerHouse_1 (EK1122)^Term 42 (EK1100)^Term 44 (EL1809)^Channel 9^Input} *)
	STP.M200A4A_MixerR4_RunStat AT %IX37.7 : BOOL;	(*  ~ {LinkedWith:TIID^C6920 (EtherCAT)^ScadaRoom_KouplerUTP (EK1100)^ScadaRoom_KouplerFiber (EK1521)^BlowerHouse_2 (EK1501)^BlowerHouse_1 (EK1122)^Term 42 (EK1100)^Term 44 (EL1809)^Channel 10^Input} *)
	STP.M200A4B_MixerR4_RunStat AT %IX38.0 : BOOL;	(*  ~ {LinkedWith:TIID^C6920 (EtherCAT)^ScadaRoom_KouplerUTP (EK1100)^ScadaRoom_KouplerFiber (EK1521)^BlowerHouse_2 (EK1501)^BlowerHouse_1 (EK1122)^Term 42 (EK1100)^Term 44 (EL1809)^Channel 11^Input} *)
	STP.M200A4C_MixerR4_RunStat AT %IX38.1 : BOOL;	(*  ~ {LinkedWith:TIID^C6920 (EtherCAT)^ScadaRoom_KouplerUTP (EK1100)^ScadaRoom_KouplerFiber (EK1521)^BlowerHouse_2 (EK1501)^BlowerHouse_1 (EK1122)^Term 42 (EK1100)^Term 44 (EL1809)^Channel 12^Input} *)
	STP.B201A1_AirBlowerS1_RunStat AT %IX144.0 : BOOL;	(*  ~ {LinkedWith:TIID^C6920 (EtherCAT)^ScadaRoom_KouplerUTP (EK1100)^ScadaRoom_KouplerFiber (EK1521)^BlowerHouse_2 (EK1501)^BlowerHouse_1 (EK1122)^Term 42 (EK1100)^Term 44 (EL1809)^Channel 13^Input} *)
	STP.B201A2_AirBlowerS1_RunStat AT %IX38.3 : BOOL;	(*  ~ {LinkedWith:TIID^C6920 (EtherCAT)^ScadaRoom_KouplerUTP (EK1100)^ScadaRoom_KouplerFiber (EK1521)^BlowerHouse_2 (EK1501)^BlowerHouse_1 (EK1122)^Term 42 (EK1100)^Term 44 (EL1809)^Channel 14^Input} *)
	STP.B201A3_AirBlowerS1_RunStat AT %IX38.4 : BOOL;	(*  ~ {LinkedWith:TIID^C6920 (EtherCAT)^ScadaRoom_KouplerUTP (EK1100)^ScadaRoom_KouplerFiber (EK1521)^BlowerHouse_2 (EK1501)^BlowerHouse_1 (EK1122)^Term 42 (EK1100)^Term 44 (EL1809)^Channel 15^Input} *)
	STP.M200A1A_MixerR1_LocalRemoteStat AT %IX38.5 : BOOL;	(*  ~ {LinkedWith:TIID^C6920 (EtherCAT)^ScadaRoom_KouplerUTP (EK1100)^ScadaRoom_KouplerFiber (EK1521)^BlowerHouse_2 (EK1501)^BlowerHouse_1 (EK1122)^Term 42 (EK1100)^Term 45 (EL1809)^Channel 1^Input} *)
	STP.M200A1B_MixerR1_LocalRemoteStat AT %IX38.6 : BOOL;	(*  ~ {LinkedWith:TIID^C6920 (EtherCAT)^ScadaRoom_KouplerUTP (EK1100)^ScadaRoom_KouplerFiber (EK1521)^BlowerHouse_2 (EK1501)^BlowerHouse_1 (EK1122)^Term 42 (EK1100)^Term 45 (EL1809)^Channel 2^Input} *)
	STP.M200A1C_MixerR1_LocalRemoteStat AT %IX38.7 : BOOL;	(*  ~ {LinkedWith:TIID^C6920 (EtherCAT)^ScadaRoom_KouplerUTP (EK1100)^ScadaRoom_KouplerFiber (EK1521)^BlowerHouse_2 (EK1501)^BlowerHouse_1 (EK1122)^Term 42 (EK1100)^Term 45 (EL1809)^Channel 3^Input} *)
	STP.M200A2A_MixerR2_LocalRemoteStat AT %IX39.0 : BOOL;	(*  ~ {LinkedWith:TIID^C6920 (EtherCAT)^ScadaRoom_KouplerUTP (EK1100)^ScadaRoom_KouplerFiber (EK1521)^BlowerHouse_2 (EK1501)^BlowerHouse_1 (EK1122)^Term 42 (EK1100)^Term 45 (EL1809)^Channel 4^Input} *)
	STP.M200A2B_MixerR2_LocalRemoteStat AT %IX39.1 : BOOL;	(*  ~ {LinkedWith:TIID^C6920 (EtherCAT)^ScadaRoom_KouplerUTP (EK1100)^ScadaRoom_KouplerFiber (EK1521)^BlowerHouse_2 (EK1501)^BlowerHouse_1 (EK1122)^Term 42 (EK1100)^Term 45 (EL1809)^Channel 5^Input} *)
	STP.M200A2C_MixerR2_LocalRemoteStat AT %IX39.2 : BOOL;	(*  ~ {LinkedWith:TIID^C6920 (EtherCAT)^ScadaRoom_KouplerUTP (EK1100)^ScadaRoom_KouplerFiber (EK1521)^BlowerHouse_2 (EK1501)^BlowerHouse_1 (EK1122)^Term 42 (EK1100)^Term 45 (EL1809)^Channel 6^Input} *)
	STP.M200A3A_MixerR3_LocalRemoteStat AT %IX39.3 : BOOL;	(*  ~ {LinkedWith:TIID^C6920 (EtherCAT)^ScadaRoom_KouplerUTP (EK1100)^ScadaRoom_KouplerFiber (EK1521)^BlowerHouse_2 (EK1501)^BlowerHouse_1 (EK1122)^Term 42 (EK1100)^Term 45 (EL1809)^Channel 7^Input} *)
	STP.M200A3B_MixerR3_LocalRemoteStat AT %IX39.4 : BOOL;	(*  ~ {LinkedWith:TIID^C6920 (EtherCAT)^ScadaRoom_KouplerUTP (EK1100)^ScadaRoom_KouplerFiber (EK1521)^BlowerHouse_2 (EK1501)^BlowerHouse_1 (EK1122)^Term 42 (EK1100)^Term 45 (EL1809)^Channel 8^Input} *)
	STP.M200A3C_MixerR3_LocalRemoteStat AT %IX39.5 : BOOL;	(*  ~ {LinkedWith:TIID^C6920 (EtherCAT)^ScadaRoom_KouplerUTP (EK1100)^ScadaRoom_KouplerFiber (EK1521)^BlowerHouse_2 (EK1501)^BlowerHouse_1 (EK1122)^Term 42 (EK1100)^Term 45 (EL1809)^Channel 9^Input} *)
	STP.M200A4A_MixerR4_LocalRemoteStat AT %IX39.6 : BOOL;	(*  ~ {LinkedWith:TIID^C6920 (EtherCAT)^ScadaRoom_KouplerUTP (EK1100)^ScadaRoom_KouplerFiber (EK1521)^BlowerHouse_2 (EK1501)^BlowerHouse_1 (EK1122)^Term 42 (EK1100)^Term 45 (EL1809)^Channel 10^Input} *)
	STP.M200A4B_MixerR4_LocalRemoteStat AT %IX39.7 : BOOL;	(*  ~ {LinkedWith:TIID^C6920 (EtherCAT)^ScadaRoom_KouplerUTP (EK1100)^ScadaRoom_KouplerFiber (EK1521)^BlowerHouse_2 (EK1501)^BlowerHouse_1 (EK1122)^Term 42 (EK1100)^Term 45 (EL1809)^Channel 11^Input} *)
	STP.M200A4C_MixerR4_LocalRemoteStat AT %IX40.0 : BOOL;	(*  ~ {LinkedWith:TIID^C6920 (EtherCAT)^ScadaRoom_KouplerUTP (EK1100)^ScadaRoom_KouplerFiber (EK1521)^BlowerHouse_2 (EK1501)^BlowerHouse_1 (EK1122)^Term 42 (EK1100)^Term 45 (EL1809)^Channel 12^Input} *)
	STP.B201A1_AirBlowerS1_LocalRemoteStat AT %IX148.0 : BOOL;	(*  ~ {LinkedWith:TIID^C6920 (EtherCAT)^ScadaRoom_KouplerUTP (EK1100)^ScadaRoom_KouplerFiber (EK1521)^BlowerHouse_2 (EK1501)^BlowerHouse_1 (EK1122)^Term 42 (EK1100)^Term 46 (EL1809)^Channel 1^Input} *)
	STP.B201A2_AirBlowerS1_LocalRemoteStat AT %IX40.2 : BOOL;	(*  ~ {LinkedWith:TIID^C6920 (EtherCAT)^ScadaRoom_KouplerUTP (EK1100)^ScadaRoom_KouplerFiber (EK1521)^BlowerHouse_2 (EK1501)^BlowerHouse_1 (EK1122)^Term 42 (EK1100)^Term 46 (EL1809)^Channel 2^Input} *)
	STP.B201A3_AirBlowerS1_LocalRemoteStat AT %IX40.3 : BOOL;	(*  ~ {LinkedWith:TIID^C6920 (EtherCAT)^ScadaRoom_KouplerUTP (EK1100)^ScadaRoom_KouplerFiber (EK1521)^BlowerHouse_2 (EK1501)^BlowerHouse_1 (EK1122)^Term 42 (EK1100)^Term 46 (EL1809)^Channel 3^Input} *)
	STP.XV261A_DecanterR1_LocalRemoteStat AT %IX40.4 : BOOL;	(*  ~ {LinkedWith:TIID^C6920 (EtherCAT)^ScadaRoom_KouplerUTP (EK1100)^ScadaRoom_KouplerFiber (EK1521)^BlowerHouse_2 (EK1501)^BlowerHouse_1 (EK1122)^Term 42 (EK1100)^Term 46 (EL1809)^Channel 4^Input} *)
	STP.XV262A_DecanterR2_LocalRemoteStat AT %IX40.5 : BOOL;	(*  ~ {LinkedWith:TIID^C6920 (EtherCAT)^ScadaRoom_KouplerUTP (EK1100)^ScadaRoom_KouplerFiber (EK1521)^BlowerHouse_2 (EK1501)^BlowerHouse_1 (EK1122)^Term 42 (EK1100)^Term 46 (EL1809)^Channel 5^Input} *)
	STP.XV263A_DecanterR3_LocalRemoteStat AT %IX40.6 : BOOL;	(*  ~ {LinkedWith:TIID^C6920 (EtherCAT)^ScadaRoom_KouplerUTP (EK1100)^ScadaRoom_KouplerFiber (EK1521)^BlowerHouse_2 (EK1501)^BlowerHouse_1 (EK1122)^Term 42 (EK1100)^Term 46 (EL1809)^Channel 6^Input} *)
	STP.XV264A_DecanterR4_LocalRemoteStat AT %IX40.7 : BOOL;	(*  ~ {LinkedWith:TIID^C6920 (EtherCAT)^ScadaRoom_KouplerUTP (EK1100)^ScadaRoom_KouplerFiber (EK1521)^BlowerHouse_2 (EK1501)^BlowerHouse_1 (EK1122)^Term 42 (EK1100)^Term 46 (EL1809)^Channel 7^Input} *)
	STP.P201A1_DesludgePumpS1_LocalRemoteStat AT %IX41.0 : BOOL;	(*  ~ {LinkedWith:TIID^C6920 (EtherCAT)^ScadaRoom_KouplerUTP (EK1100)^ScadaRoom_KouplerFiber (EK1521)^BlowerHouse_2 (EK1501)^BlowerHouse_1 (EK1122)^Term 42 (EK1100)^Term 46 (EL1809)^Channel 8^Input} *)
	STP.P201A2_DesludgePumpS1_LocalRemoteStat AT %IX41.1 : BOOL;	(*  ~ {LinkedWith:TIID^C6920 (EtherCAT)^ScadaRoom_KouplerUTP (EK1100)^ScadaRoom_KouplerFiber (EK1521)^BlowerHouse_2 (EK1501)^BlowerHouse_1 (EK1122)^Term 42 (EK1100)^Term 46 (EL1809)^Channel 9^Input} *)
	STP.P201A1_DesludgePumpS1_RunStat AT %IX41.2 : BOOL;	(*  ~ {LinkedWith:TIID^C6920 (EtherCAT)^ScadaRoom_KouplerUTP (EK1100)^ScadaRoom_KouplerFiber (EK1521)^BlowerHouse_2 (EK1501)^BlowerHouse_1 (EK1122)^Term 42 (EK1100)^Term 46 (EL1809)^Channel 10^Input} *)
	STP.P201A2_DesludgePumpS1_RunStat AT %IX41.3 : BOOL;	(*  ~ {LinkedWith:TIID^C6920 (EtherCAT)^ScadaRoom_KouplerUTP (EK1100)^ScadaRoom_KouplerFiber (EK1521)^BlowerHouse_2 (EK1501)^BlowerHouse_1 (EK1122)^Term 42 (EK1100)^Term 46 (EL1809)^Channel 11^Input} *)
	STP.M200A1A_MixerR1_OverloadStat AT %IX41.4 : BOOL;	(*  ~ {LinkedWith:TIID^C6920 (EtherCAT)^ScadaRoom_KouplerUTP (EK1100)^ScadaRoom_KouplerFiber (EK1521)^BlowerHouse_2 (EK1501)^BlowerHouse_1 (EK1122)^Term 42 (EK1100)^Term 47 (EL1809)^Channel 1^Input} *)
	STP.M200A1A_MixerR1_IncompleteStat AT %IX41.5 : BOOL;	(*  ~ {LinkedWith:TIID^C6920 (EtherCAT)^ScadaRoom_KouplerUTP (EK1100)^ScadaRoom_KouplerFiber (EK1521)^BlowerHouse_2 (EK1501)^BlowerHouse_1 (EK1122)^Term 42 (EK1100)^Term 47 (EL1809)^Channel 2^Input} *)
	STP.M200A1B_MixerR1_OverloadStat AT %IX41.6 : BOOL;	(*  ~ {LinkedWith:TIID^C6920 (EtherCAT)^ScadaRoom_KouplerUTP (EK1100)^ScadaRoom_KouplerFiber (EK1521)^BlowerHouse_2 (EK1501)^BlowerHouse_1 (EK1122)^Term 42 (EK1100)^Term 47 (EL1809)^Channel 3^Input} *)
	STP.M200A1B_MixerR1_IncompleteStat AT %IX41.7 : BOOL;	(*  ~ {LinkedWith:TIID^C6920 (EtherCAT)^ScadaRoom_KouplerUTP (EK1100)^ScadaRoom_KouplerFiber (EK1521)^BlowerHouse_2 (EK1501)^BlowerHouse_1 (EK1122)^Term 42 (EK1100)^Term 47 (EL1809)^Channel 4^Input} *)
	STP.M200A1C_MixerR1_OverloadStat AT %IX42.0 : BOOL;	(*  ~ {LinkedWith:TIID^C6920 (EtherCAT)^ScadaRoom_KouplerUTP (EK1100)^ScadaRoom_KouplerFiber (EK1521)^BlowerHouse_2 (EK1501)^BlowerHouse_1 (EK1122)^Term 42 (EK1100)^Term 47 (EL1809)^Channel 5^Input} *)
	STP.M200A1C_MixerR1_IncompleteStat AT %IX42.1 : BOOL;	(*  ~ {LinkedWith:TIID^C6920 (EtherCAT)^ScadaRoom_KouplerUTP (EK1100)^ScadaRoom_KouplerFiber (EK1521)^BlowerHouse_2 (EK1501)^BlowerHouse_1 (EK1122)^Term 42 (EK1100)^Term 47 (EL1809)^Channel 6^Input} *)
	STP.M200A2A_MixerR2_OverloadStat AT %IX42.2 : BOOL;	(*  ~ {LinkedWith:TIID^C6920 (EtherCAT)^ScadaRoom_KouplerUTP (EK1100)^ScadaRoom_KouplerFiber (EK1521)^BlowerHouse_2 (EK1501)^BlowerHouse_1 (EK1122)^Term 42 (EK1100)^Term 47 (EL1809)^Channel 7^Input} *)
	STP.M200A2A_MixerR2_IncompleteStat AT %IX42.3 : BOOL;	(*  ~ {LinkedWith:TIID^C6920 (EtherCAT)^ScadaRoom_KouplerUTP (EK1100)^ScadaRoom_KouplerFiber (EK1521)^BlowerHouse_2 (EK1501)^BlowerHouse_1 (EK1122)^Term 42 (EK1100)^Term 47 (EL1809)^Channel 8^Input} *)
	STP.M200A2B_MixerR2_OverloadStat AT %IX42.4 : BOOL;	(*  ~ {LinkedWith:TIID^C6920 (EtherCAT)^ScadaRoom_KouplerUTP (EK1100)^ScadaRoom_KouplerFiber (EK1521)^BlowerHouse_2 (EK1501)^BlowerHouse_1 (EK1122)^Term 42 (EK1100)^Term 47 (EL1809)^Channel 9^Input} *)
	STP.M200A2B_MixerR2_IncompleteStat AT %IX42.5 : BOOL;	(*  ~ {LinkedWith:TIID^C6920 (EtherCAT)^ScadaRoom_KouplerUTP (EK1100)^ScadaRoom_KouplerFiber (EK1521)^BlowerHouse_2 (EK1501)^BlowerHouse_1 (EK1122)^Term 42 (EK1100)^Term 47 (EL1809)^Channel 10^Input} *)
	STP.M200A2C_MixerR2_OverloadStat AT %IX42.6 : BOOL;	(*  ~ {LinkedWith:TIID^C6920 (EtherCAT)^ScadaRoom_KouplerUTP (EK1100)^ScadaRoom_KouplerFiber (EK1521)^BlowerHouse_2 (EK1501)^BlowerHouse_1 (EK1122)^Term 42 (EK1100)^Term 47 (EL1809)^Channel 11^Input} *)
	STP.M200A2C_MixerR2_IncompleteStat AT %IX42.7 : BOOL;	(*  ~ {LinkedWith:TIID^C6920 (EtherCAT)^ScadaRoom_KouplerUTP (EK1100)^ScadaRoom_KouplerFiber (EK1521)^BlowerHouse_2 (EK1501)^BlowerHouse_1 (EK1122)^Term 42 (EK1100)^Term 47 (EL1809)^Channel 12^Input} *)
	STP.M200A3A_MixerR3_OverloadStat AT %IX43.0 : BOOL;	(*  ~ {LinkedWith:TIID^C6920 (EtherCAT)^ScadaRoom_KouplerUTP (EK1100)^ScadaRoom_KouplerFiber (EK1521)^BlowerHouse_2 (EK1501)^BlowerHouse_1 (EK1122)^Term 42 (EK1100)^Term 47 (EL1809)^Channel 13^Input} *)
	STP.M200A3A_MixerR3_IncompleteStat AT %IX43.1 : BOOL;	(*  ~ {LinkedWith:TIID^C6920 (EtherCAT)^ScadaRoom_KouplerUTP (EK1100)^ScadaRoom_KouplerFiber (EK1521)^BlowerHouse_2 (EK1501)^BlowerHouse_1 (EK1122)^Term 42 (EK1100)^Term 47 (EL1809)^Channel 14^Input} *)
	STP.M200A3B_MixerR3_OverloadStat AT %IX43.2 : BOOL;	(*  ~ {LinkedWith:TIID^C6920 (EtherCAT)^ScadaRoom_KouplerUTP (EK1100)^ScadaRoom_KouplerFiber (EK1521)^BlowerHouse_2 (EK1501)^BlowerHouse_1 (EK1122)^Term 42 (EK1100)^Term 47 (EL1809)^Channel 15^Input} *)
	STP.M200A3B_MixerR3_IncompleteStat AT %IX43.3 : BOOL;	(*  ~ {LinkedWith:TIID^C6920 (EtherCAT)^ScadaRoom_KouplerUTP (EK1100)^ScadaRoom_KouplerFiber (EK1521)^BlowerHouse_2 (EK1501)^BlowerHouse_1 (EK1122)^Term 42 (EK1100)^Term 47 (EL1809)^Channel 16^Input} *)
	STP.M200A3C_MixerR3_OverloadStat AT %IX43.4 : BOOL;	(*  ~ {LinkedWith:TIID^C6920 (EtherCAT)^ScadaRoom_KouplerUTP (EK1100)^ScadaRoom_KouplerFiber (EK1521)^BlowerHouse_2 (EK1501)^BlowerHouse_1 (EK1122)^Term 42 (EK1100)^Term 48 (EL1809)^Channel 1^Input} *)
	STP.M200A3C_MixerR3_IncompleteStat AT %IX43.5 : BOOL;	(*  ~ {LinkedWith:TIID^C6920 (EtherCAT)^ScadaRoom_KouplerUTP (EK1100)^ScadaRoom_KouplerFiber (EK1521)^BlowerHouse_2 (EK1501)^BlowerHouse_1 (EK1122)^Term 42 (EK1100)^Term 48 (EL1809)^Channel 2^Input} *)
	STP.M200A4A_MixerR4_OverloadStat AT %IX43.6 : BOOL;	(*  ~ {LinkedWith:TIID^C6920 (EtherCAT)^ScadaRoom_KouplerUTP (EK1100)^ScadaRoom_KouplerFiber (EK1521)^BlowerHouse_2 (EK1501)^BlowerHouse_1 (EK1122)^Term 42 (EK1100)^Term 48 (EL1809)^Channel 3^Input} *)
	STP.M200A4A_MixerR4_IncompleteStat AT %IX43.7 : BOOL;	(*  ~ {LinkedWith:TIID^C6920 (EtherCAT)^ScadaRoom_KouplerUTP (EK1100)^ScadaRoom_KouplerFiber (EK1521)^BlowerHouse_2 (EK1501)^BlowerHouse_1 (EK1122)^Term 42 (EK1100)^Term 48 (EL1809)^Channel 4^Input} *)
	STP.M200A4B_MixerR4_OverloadStat AT %IX44.0 : BOOL;	(*  ~ {LinkedWith:TIID^C6920 (EtherCAT)^ScadaRoom_KouplerUTP (EK1100)^ScadaRoom_KouplerFiber (EK1521)^BlowerHouse_2 (EK1501)^BlowerHouse_1 (EK1122)^Term 42 (EK1100)^Term 48 (EL1809)^Channel 5^Input} *)
	STP.M200A4B_MixerR4_IncompleteStat AT %IX44.1 : BOOL;	(*  ~ {LinkedWith:TIID^C6920 (EtherCAT)^ScadaRoom_KouplerUTP (EK1100)^ScadaRoom_KouplerFiber (EK1521)^BlowerHouse_2 (EK1501)^BlowerHouse_1 (EK1122)^Term 42 (EK1100)^Term 48 (EL1809)^Channel 6^Input} *)
	STP.M200A4C_MixerR4_OverloadStat AT %IX44.2 : BOOL;	(*  ~ {LinkedWith:TIID^C6920 (EtherCAT)^ScadaRoom_KouplerUTP (EK1100)^ScadaRoom_KouplerFiber (EK1521)^BlowerHouse_2 (EK1501)^BlowerHouse_1 (EK1122)^Term 42 (EK1100)^Term 48 (EL1809)^Channel 7^Input} *)
	STP.M200A4C_MixerR4_IncompleteStat AT %IX44.3 : BOOL;	(*  ~ {LinkedWith:TIID^C6920 (EtherCAT)^ScadaRoom_KouplerUTP (EK1100)^ScadaRoom_KouplerFiber (EK1521)^BlowerHouse_2 (EK1501)^BlowerHouse_1 (EK1122)^Term 42 (EK1100)^Term 48 (EL1809)^Channel 8^Input} *)
	STP.B201A1_AirBlowerS1_OverloadStat AT %IX44.4 : BOOL;	(*  ~ {LinkedWith:TIID^C6920 (EtherCAT)^ScadaRoom_KouplerUTP (EK1100)^ScadaRoom_KouplerFiber (EK1521)^BlowerHouse_2 (EK1501)^BlowerHouse_1 (EK1122)^Term 42 (EK1100)^Term 48 (EL1809)^Channel 9^Input} *)
	STP.B201A1_AirBlowerS1_IncompleteStat AT %IX44.5 : BOOL;	(*  ~ {LinkedWith:TIID^C6920 (EtherCAT)^ScadaRoom_KouplerUTP (EK1100)^ScadaRoom_KouplerFiber (EK1521)^BlowerHouse_2 (EK1501)^BlowerHouse_1 (EK1122)^Term 42 (EK1100)^Term 48 (EL1809)^Channel 10^Input} *)
	STP.B201A2_AirBlowerS1_OverloadStat AT %IX44.6 : BOOL;	(*  ~ {LinkedWith:TIID^C6920 (EtherCAT)^ScadaRoom_KouplerUTP (EK1100)^ScadaRoom_KouplerFiber (EK1521)^BlowerHouse_2 (EK1501)^BlowerHouse_1 (EK1122)^Term 42 (EK1100)^Term 48 (EL1809)^Channel 11^Input} *)
	STP.B201A2_AirBlowerS1_IncompleteStat AT %IX44.7 : BOOL;	(*  ~ {LinkedWith:TIID^C6920 (EtherCAT)^ScadaRoom_KouplerUTP (EK1100)^ScadaRoom_KouplerFiber (EK1521)^BlowerHouse_2 (EK1501)^BlowerHouse_1 (EK1122)^Term 42 (EK1100)^Term 48 (EL1809)^Channel 12^Input} *)
	STP.B201A3_AirBlowerS1_OverloadStat AT %IX45.0 : BOOL;	(*  ~ {LinkedWith:TIID^C6920 (EtherCAT)^ScadaRoom_KouplerUTP (EK1100)^ScadaRoom_KouplerFiber (EK1521)^BlowerHouse_2 (EK1501)^BlowerHouse_1 (EK1122)^Term 42 (EK1100)^Term 48 (EL1809)^Channel 13^Input} *)
	STP.B201A3_AirBlowerS1_IncompleteStat AT %IX45.1 : BOOL;	(*  ~ {LinkedWith:TIID^C6920 (EtherCAT)^ScadaRoom_KouplerUTP (EK1100)^ScadaRoom_KouplerFiber (EK1521)^BlowerHouse_2 (EK1501)^BlowerHouse_1 (EK1122)^Term 42 (EK1100)^Term 48 (EL1809)^Channel 14^Input} *)
	STP.P201A1_DesludgePumpS1_OverloadStatus AT %IX45.2 : BOOL;	(*  ~ {LinkedWith:TIID^C6920 (EtherCAT)^ScadaRoom_KouplerUTP (EK1100)^ScadaRoom_KouplerFiber (EK1521)^BlowerHouse_2 (EK1501)^BlowerHouse_1 (EK1122)^Term 42 (EK1100)^Term 48 (EL1809)^Channel 15^Input} *)
	STP.P201A2_DesludgePumpS1_OverloadStatus AT %IX45.3 : BOOL;	(*  ~ {LinkedWith:TIID^C6920 (EtherCAT)^ScadaRoom_KouplerUTP (EK1100)^ScadaRoom_KouplerFiber (EK1521)^BlowerHouse_2 (EK1501)^BlowerHouse_1 (EK1122)^Term 42 (EK1100)^Term 48 (EL1809)^Channel 16^Input} *)
	STP.M200A1A_MixerR1_EStopStat AT %IX45.4 : BOOL;	(*  ~ {LinkedWith:TIID^C6920 (EtherCAT)^ScadaRoom_KouplerUTP (EK1100)^ScadaRoom_KouplerFiber (EK1521)^BlowerHouse_2 (EK1501)^BlowerHouse_1 (EK1122)^Term 42 (EK1100)^Term 49 (EL1809)^Channel 1^Input} *)
	STP.M200A1B_MixerR1_EStopStat AT %IX45.5 : BOOL;	(*  ~ {LinkedWith:TIID^C6920 (EtherCAT)^ScadaRoom_KouplerUTP (EK1100)^ScadaRoom_KouplerFiber (EK1521)^BlowerHouse_2 (EK1501)^BlowerHouse_1 (EK1122)^Term 42 (EK1100)^Term 49 (EL1809)^Channel 2^Input} *)
	STP.M200A1C_MixerR1_EStopStat AT %IX45.6 : BOOL;	(*  ~ {LinkedWith:TIID^C6920 (EtherCAT)^ScadaRoom_KouplerUTP (EK1100)^ScadaRoom_KouplerFiber (EK1521)^BlowerHouse_2 (EK1501)^BlowerHouse_1 (EK1122)^Term 42 (EK1100)^Term 49 (EL1809)^Channel 3^Input} *)
	STP.M200A2A_MixerR2_EStopStat AT %IX45.7 : BOOL;	(*  ~ {LinkedWith:TIID^C6920 (EtherCAT)^ScadaRoom_KouplerUTP (EK1100)^ScadaRoom_KouplerFiber (EK1521)^BlowerHouse_2 (EK1501)^BlowerHouse_1 (EK1122)^Term 42 (EK1100)^Term 49 (EL1809)^Channel 4^Input} *)
	STP.M200A2B_MixerR2_EStopStat AT %IX46.0 : BOOL;	(*  ~ {LinkedWith:TIID^C6920 (EtherCAT)^ScadaRoom_KouplerUTP (EK1100)^ScadaRoom_KouplerFiber (EK1521)^BlowerHouse_2 (EK1501)^BlowerHouse_1 (EK1122)^Term 42 (EK1100)^Term 49 (EL1809)^Channel 5^Input} *)
	STP.M200A2C_MixerR2_EStopStat AT %IX46.1 : BOOL;	(*  ~ {LinkedWith:TIID^C6920 (EtherCAT)^ScadaRoom_KouplerUTP (EK1100)^ScadaRoom_KouplerFiber (EK1521)^BlowerHouse_2 (EK1501)^BlowerHouse_1 (EK1122)^Term 42 (EK1100)^Term 49 (EL1809)^Channel 6^Input} *)
	STP.M200A3A_MixerR3_EStopStat AT %IX46.2 : BOOL;	(*  ~ {LinkedWith:TIID^C6920 (EtherCAT)^ScadaRoom_KouplerUTP (EK1100)^ScadaRoom_KouplerFiber (EK1521)^BlowerHouse_2 (EK1501)^BlowerHouse_1 (EK1122)^Term 42 (EK1100)^Term 49 (EL1809)^Channel 7^Input} *)
	STP.M200A3B_MixerR3_EStopStat AT %IX46.3 : BOOL;	(*  ~ {LinkedWith:TIID^C6920 (EtherCAT)^ScadaRoom_KouplerUTP (EK1100)^ScadaRoom_KouplerFiber (EK1521)^BlowerHouse_2 (EK1501)^BlowerHouse_1 (EK1122)^Term 42 (EK1100)^Term 49 (EL1809)^Channel 8^Input} *)
	STP.M200A3C_MixerR3_EStopStat AT %IX46.4 : BOOL;	(*  ~ {LinkedWith:TIID^C6920 (EtherCAT)^ScadaRoom_KouplerUTP (EK1100)^ScadaRoom_KouplerFiber (EK1521)^BlowerHouse_2 (EK1501)^BlowerHouse_1 (EK1122)^Term 42 (EK1100)^Term 49 (EL1809)^Channel 9^Input} *)
	STP.M200A4A_MixerR3_EStopStat AT %IX46.5 : BOOL;	(*  ~ {LinkedWith:TIID^C6920 (EtherCAT)^ScadaRoom_KouplerUTP (EK1100)^ScadaRoom_KouplerFiber (EK1521)^BlowerHouse_2 (EK1501)^BlowerHouse_1 (EK1122)^Term 42 (EK1100)^Term 49 (EL1809)^Channel 10^Input} *)
	STP.M200A4B_MixerR3_EStopStat AT %IX46.6 : BOOL;	(*  ~ {LinkedWith:TIID^C6920 (EtherCAT)^ScadaRoom_KouplerUTP (EK1100)^ScadaRoom_KouplerFiber (EK1521)^BlowerHouse_2 (EK1501)^BlowerHouse_1 (EK1122)^Term 42 (EK1100)^Term 49 (EL1809)^Channel 11^Input} *)
	STP.M200A4C_MixerR3_EStopStat AT %IX46.7 : BOOL;	(*  ~ {LinkedWith:TIID^C6920 (EtherCAT)^ScadaRoom_KouplerUTP (EK1100)^ScadaRoom_KouplerFiber (EK1521)^BlowerHouse_2 (EK1501)^BlowerHouse_1 (EK1122)^Term 42 (EK1100)^Term 49 (EL1809)^Channel 12^Input} *)
	STP.B201A1_AirBlowerS1_EStopStat AT %IX47.0 : BOOL;	(*  ~ {LinkedWith:TIID^C6920 (EtherCAT)^ScadaRoom_KouplerUTP (EK1100)^ScadaRoom_KouplerFiber (EK1521)^BlowerHouse_2 (EK1501)^BlowerHouse_1 (EK1122)^Term 42 (EK1100)^Term 50 (EL1809)^Channel 1^Input} *)
	STP.B201A2_AirBlowerS1_EStopStat AT %IX47.1 : BOOL;	(*  ~ {LinkedWith:TIID^C6920 (EtherCAT)^ScadaRoom_KouplerUTP (EK1100)^ScadaRoom_KouplerFiber (EK1521)^BlowerHouse_2 (EK1501)^BlowerHouse_1 (EK1122)^Term 42 (EK1100)^Term 50 (EL1809)^Channel 2^Input} *)
	STP.B201A3_AirBlowerS1_EStopStat AT %IX47.2 : BOOL;	(*  ~ {LinkedWith:TIID^C6920 (EtherCAT)^ScadaRoom_KouplerUTP (EK1100)^ScadaRoom_KouplerFiber (EK1521)^BlowerHouse_2 (EK1501)^BlowerHouse_1 (EK1122)^Term 42 (EK1100)^Term 50 (EL1809)^Channel 3^Input} *)
	STP.XV261A_DecanterR1_EStopStat AT %IX47.3 : BOOL;	(*  ~ {LinkedWith:TIID^C6920 (EtherCAT)^ScadaRoom_KouplerUTP (EK1100)^ScadaRoom_KouplerFiber (EK1521)^BlowerHouse_2 (EK1501)^BlowerHouse_1 (EK1122)^Term 42 (EK1100)^Term 50 (EL1809)^Channel 4^Input} *)
	STP.XV262A_DecanterR2_EStopStat AT %IX47.4 : BOOL;	(*  ~ {LinkedWith:TIID^C6920 (EtherCAT)^ScadaRoom_KouplerUTP (EK1100)^ScadaRoom_KouplerFiber (EK1521)^BlowerHouse_2 (EK1501)^BlowerHouse_1 (EK1122)^Term 42 (EK1100)^Term 50 (EL1809)^Channel 5^Input} *)
	STP.XV263A_DecanterR3_EStopStat AT %IX47.5 : BOOL;	(*  ~ {LinkedWith:TIID^C6920 (EtherCAT)^ScadaRoom_KouplerUTP (EK1100)^ScadaRoom_KouplerFiber (EK1521)^BlowerHouse_2 (EK1501)^BlowerHouse_1 (EK1122)^Term 42 (EK1100)^Term 50 (EL1809)^Channel 6^Input} *)
	STP.XV264A_DecanterR4_EStopStat AT %IX47.6 : BOOL;	(*  ~ {LinkedWith:TIID^C6920 (EtherCAT)^ScadaRoom_KouplerUTP (EK1100)^ScadaRoom_KouplerFiber (EK1521)^BlowerHouse_2 (EK1501)^BlowerHouse_1 (EK1122)^Term 42 (EK1100)^Term 50 (EL1809)^Channel 7^Input} *)
	STP.P201A1_DesludgePumpS1_EStopStat AT %IX47.7 : BOOL;	(*  ~ {LinkedWith:TIID^C6920 (EtherCAT)^ScadaRoom_KouplerUTP (EK1100)^ScadaRoom_KouplerFiber (EK1521)^BlowerHouse_2 (EK1501)^BlowerHouse_1 (EK1122)^Term 42 (EK1100)^Term 50 (EL1809)^Channel 8^Input} *)
	STP.P201A2_DesludgePumpS1_EStopStat AT %IX48.0 : BOOL;	(*  ~ {LinkedWith:TIID^C6920 (EtherCAT)^ScadaRoom_KouplerUTP (EK1100)^ScadaRoom_KouplerFiber (EK1521)^BlowerHouse_2 (EK1501)^BlowerHouse_1 (EK1122)^Term 42 (EK1100)^Term 50 (EL1809)^Channel 9^Input} *)
	STP.XV261A_DecanterR1_FwdStat AT %IX48.1 : BOOL;	(*  ~ {LinkedWith:TIID^C6920 (EtherCAT)^ScadaRoom_KouplerUTP (EK1100)^ScadaRoom_KouplerFiber (EK1521)^BlowerHouse_2 (EK1501)^BlowerHouse_1 (EK1122)^Term 42 (EK1100)^Term 51 (EL1809)^Channel 1^Input} *)
	STP.XV262A_DecanterR2_FwdStat AT %IX48.2 : BOOL;	(*  ~ {LinkedWith:TIID^C6920 (EtherCAT)^ScadaRoom_KouplerUTP (EK1100)^ScadaRoom_KouplerFiber (EK1521)^BlowerHouse_2 (EK1501)^BlowerHouse_1 (EK1122)^Term 42 (EK1100)^Term 51 (EL1809)^Channel 2^Input} *)
	STP.XV263A_DecanterR3_FwdStat AT %IX48.3 : BOOL;	(*  ~ {LinkedWith:TIID^C6920 (EtherCAT)^ScadaRoom_KouplerUTP (EK1100)^ScadaRoom_KouplerFiber (EK1521)^BlowerHouse_2 (EK1501)^BlowerHouse_1 (EK1122)^Term 42 (EK1100)^Term 51 (EL1809)^Channel 3^Input} *)
	STP.XV264A_DecanterR4_FwdStat AT %IX48.4 : BOOL;	(*  ~ {LinkedWith:TIID^C6920 (EtherCAT)^ScadaRoom_KouplerUTP (EK1100)^ScadaRoom_KouplerFiber (EK1521)^BlowerHouse_2 (EK1501)^BlowerHouse_1 (EK1122)^Term 42 (EK1100)^Term 51 (EL1809)^Channel 4^Input} *)
	STP.XV261A_DecanterR1_RvsStat AT %IX48.5 : BOOL;	(*  ~ {LinkedWith:TIID^C6920 (EtherCAT)^ScadaRoom_KouplerUTP (EK1100)^ScadaRoom_KouplerFiber (EK1521)^BlowerHouse_2 (EK1501)^BlowerHouse_1 (EK1122)^Term 42 (EK1100)^Term 51 (EL1809)^Channel 5^Input} *)
	STP.XV262A_DecanterR2_RvsStat AT %IX48.6 : BOOL;	(*  ~ {LinkedWith:TIID^C6920 (EtherCAT)^ScadaRoom_KouplerUTP (EK1100)^ScadaRoom_KouplerFiber (EK1521)^BlowerHouse_2 (EK1501)^BlowerHouse_1 (EK1122)^Term 42 (EK1100)^Term 51 (EL1809)^Channel 6^Input} *)
	STP.XV263A_DecanterR3_RvsStat AT %IX48.7 : BOOL;	(*  ~ {LinkedWith:TIID^C6920 (EtherCAT)^ScadaRoom_KouplerUTP (EK1100)^ScadaRoom_KouplerFiber (EK1521)^BlowerHouse_2 (EK1501)^BlowerHouse_1 (EK1122)^Term 42 (EK1100)^Term 51 (EL1809)^Channel 7^Input} *)
	STP.XV264A_DecanterR4_RvsStat AT %IX49.0 : BOOL;	(*  ~ {LinkedWith:TIID^C6920 (EtherCAT)^ScadaRoom_KouplerUTP (EK1100)^ScadaRoom_KouplerFiber (EK1521)^BlowerHouse_2 (EK1501)^BlowerHouse_1 (EK1122)^Term 42 (EK1100)^Term 51 (EL1809)^Channel 8^Input} *)
	STP.M200A1A_MixerR1_RunCmd AT %QX12.0 : BOOL;	(*  ~ {LinkedWith:TIID^C6920 (EtherCAT)^ScadaRoom_KouplerUTP (EK1100)^ScadaRoom_KouplerFiber (EK1521)^BlowerHouse_2 (EK1501)^BlowerHouse_1 (EK1122)^Term 42 (EK1100)^Term 53 (EL2809)^Channel 1^Output} *)
	STP.M200A1B_MixerR1_RunCmd AT %QX12.1 : BOOL;	(*  ~ {LinkedWith:TIID^C6920 (EtherCAT)^ScadaRoom_KouplerUTP (EK1100)^ScadaRoom_KouplerFiber (EK1521)^BlowerHouse_2 (EK1501)^BlowerHouse_1 (EK1122)^Term 42 (EK1100)^Term 53 (EL2809)^Channel 2^Output} *)
	STP.M200A1C_MixerR1_RunCmd AT %QX12.2 : BOOL;	(*  ~ {LinkedWith:TIID^C6920 (EtherCAT)^ScadaRoom_KouplerUTP (EK1100)^ScadaRoom_KouplerFiber (EK1521)^BlowerHouse_2 (EK1501)^BlowerHouse_1 (EK1122)^Term 42 (EK1100)^Term 53 (EL2809)^Channel 3^Output} *)
	STP.M200A2A_MixerR2_RunCmd AT %QX12.3 : BOOL;	(*  ~ {LinkedWith:TIID^C6920 (EtherCAT)^ScadaRoom_KouplerUTP (EK1100)^ScadaRoom_KouplerFiber (EK1521)^BlowerHouse_2 (EK1501)^BlowerHouse_1 (EK1122)^Term 42 (EK1100)^Term 53 (EL2809)^Channel 4^Output} *)
	STP.M200A2B_MixerR2_RunCmd AT %QX12.4 : BOOL;	(*  ~ {LinkedWith:TIID^C6920 (EtherCAT)^ScadaRoom_KouplerUTP (EK1100)^ScadaRoom_KouplerFiber (EK1521)^BlowerHouse_2 (EK1501)^BlowerHouse_1 (EK1122)^Term 42 (EK1100)^Term 53 (EL2809)^Channel 5^Output} *)
	STP.M200A2C_MixerR2_RunCmd AT %QX12.5 : BOOL;	(*  ~ {LinkedWith:TIID^C6920 (EtherCAT)^ScadaRoom_KouplerUTP (EK1100)^ScadaRoom_KouplerFiber (EK1521)^BlowerHouse_2 (EK1501)^BlowerHouse_1 (EK1122)^Term 42 (EK1100)^Term 53 (EL2809)^Channel 6^Output} *)
	STP.M200A3A_MixerR3_RunCmd AT %QX12.6 : BOOL;	(*  ~ {LinkedWith:TIID^C6920 (EtherCAT)^ScadaRoom_KouplerUTP (EK1100)^ScadaRoom_KouplerFiber (EK1521)^BlowerHouse_2 (EK1501)^BlowerHouse_1 (EK1122)^Term 42 (EK1100)^Term 53 (EL2809)^Channel 7^Output} *)
	STP.M200A3B_MixerR3_RunCmd AT %QX12.7 : BOOL;	(*  ~ {LinkedWith:TIID^C6920 (EtherCAT)^ScadaRoom_KouplerUTP (EK1100)^ScadaRoom_KouplerFiber (EK1521)^BlowerHouse_2 (EK1501)^BlowerHouse_1 (EK1122)^Term 42 (EK1100)^Term 53 (EL2809)^Channel 8^Output} *)
	STP.M200A3C_MixerR3_RunCmd AT %QX13.0 : BOOL;	(*  ~ {LinkedWith:TIID^C6920 (EtherCAT)^ScadaRoom_KouplerUTP (EK1100)^ScadaRoom_KouplerFiber (EK1521)^BlowerHouse_2 (EK1501)^BlowerHouse_1 (EK1122)^Term 42 (EK1100)^Term 53 (EL2809)^Channel 9^Output} *)
	STP.M200A4A_MixerR4_RunCmd AT %QX13.1 : BOOL;	(*  ~ {LinkedWith:TIID^C6920 (EtherCAT)^ScadaRoom_KouplerUTP (EK1100)^ScadaRoom_KouplerFiber (EK1521)^BlowerHouse_2 (EK1501)^BlowerHouse_1 (EK1122)^Term 42 (EK1100)^Term 53 (EL2809)^Channel 10^Output} *)
	STP.M200A4B_MixerR4_RunCmd AT %QX13.2 : BOOL;	(*  ~ {LinkedWith:TIID^C6920 (EtherCAT)^ScadaRoom_KouplerUTP (EK1100)^ScadaRoom_KouplerFiber (EK1521)^BlowerHouse_2 (EK1501)^BlowerHouse_1 (EK1122)^Term 42 (EK1100)^Term 53 (EL2809)^Channel 11^Output} *)
	STP.M200A4C_MixerR4_RunCmd AT %QX72.2 : BOOL;	(*  ~ {LinkedWith:TIID^C6920 (EtherCAT)^ScadaRoom_KouplerUTP (EK1100)^ScadaRoom_KouplerFiber (EK1521)^BlowerHouse_2 (EK1501)^BlowerHouse_1 (EK1122)^Term 42 (EK1100)^Term 53 (EL2809)^Channel 12^Output} *)
	STP.XV261A_DecanterR1_FwdCmd AT %QX13.4 : BOOL;	(*  ~ {LinkedWith:TIID^C6920 (EtherCAT)^ScadaRoom_KouplerUTP (EK1100)^ScadaRoom_KouplerFiber (EK1521)^BlowerHouse_2 (EK1501)^BlowerHouse_1 (EK1122)^Term 42 (EK1100)^Term 54 (EL2809)^Channel 1^Output} *)
	STP.XV262A_DecanterR2_FwdCmd AT %QX13.5 : BOOL;	(*  ~ {LinkedWith:TIID^C6920 (EtherCAT)^ScadaRoom_KouplerUTP (EK1100)^ScadaRoom_KouplerFiber (EK1521)^BlowerHouse_2 (EK1501)^BlowerHouse_1 (EK1122)^Term 42 (EK1100)^Term 54 (EL2809)^Channel 2^Output} *)
	STP.XV263A_DecanterR3_FwdCmd AT %QX13.6 : BOOL;	(*  ~ {LinkedWith:TIID^C6920 (EtherCAT)^ScadaRoom_KouplerUTP (EK1100)^ScadaRoom_KouplerFiber (EK1521)^BlowerHouse_2 (EK1501)^BlowerHouse_1 (EK1122)^Term 42 (EK1100)^Term 54 (EL2809)^Channel 3^Output} *)
	STP.XV264A_DecanterR4_FwdCmd AT %QX13.7 : BOOL;	(*  ~ {LinkedWith:TIID^C6920 (EtherCAT)^ScadaRoom_KouplerUTP (EK1100)^ScadaRoom_KouplerFiber (EK1521)^BlowerHouse_2 (EK1501)^BlowerHouse_1 (EK1122)^Term 42 (EK1100)^Term 54 (EL2809)^Channel 4^Output} *)
	STP.XV261A_DecanterR1_RvsCmd AT %QX14.0 : BOOL;	(*  ~ {LinkedWith:TIID^C6920 (EtherCAT)^ScadaRoom_KouplerUTP (EK1100)^ScadaRoom_KouplerFiber (EK1521)^BlowerHouse_2 (EK1501)^BlowerHouse_1 (EK1122)^Term 42 (EK1100)^Term 54 (EL2809)^Channel 5^Output} *)
	STP.XV262A_DecanterR2_RvsCmd AT %QX14.1 : BOOL;	(*  ~ {LinkedWith:TIID^C6920 (EtherCAT)^ScadaRoom_KouplerUTP (EK1100)^ScadaRoom_KouplerFiber (EK1521)^BlowerHouse_2 (EK1501)^BlowerHouse_1 (EK1122)^Term 42 (EK1100)^Term 54 (EL2809)^Channel 6^Output} *)
	STP.XV263A_DecanterR3_RvsCmd AT %QX14.2 : BOOL;	(*  ~ {LinkedWith:TIID^C6920 (EtherCAT)^ScadaRoom_KouplerUTP (EK1100)^ScadaRoom_KouplerFiber (EK1521)^BlowerHouse_2 (EK1501)^BlowerHouse_1 (EK1122)^Term 42 (EK1100)^Term 54 (EL2809)^Channel 7^Output} *)
	STP.XV264A_DecanterR4_RvsCmd AT %QX14.3 : BOOL;	(*  ~ {LinkedWith:TIID^C6920 (EtherCAT)^ScadaRoom_KouplerUTP (EK1100)^ScadaRoom_KouplerFiber (EK1521)^BlowerHouse_2 (EK1501)^BlowerHouse_1 (EK1122)^Term 42 (EK1100)^Term 54 (EL2809)^Channel 8^Output} *)
	STP.B201A1_AirBlowerS1_RunCmd AT %QX14.4 : BOOL;	(*  ~ {LinkedWith:TIID^C6920 (EtherCAT)^ScadaRoom_KouplerUTP (EK1100)^ScadaRoom_KouplerFiber (EK1521)^BlowerHouse_2 (EK1501)^BlowerHouse_1 (EK1122)^Term 42 (EK1100)^Term 54 (EL2809)^Channel 9^Output} *)
	STP.B201A2_AirBlowerS1_RunCmd AT %QX14.5 : BOOL;	(*  ~ {LinkedWith:TIID^C6920 (EtherCAT)^ScadaRoom_KouplerUTP (EK1100)^ScadaRoom_KouplerFiber (EK1521)^BlowerHouse_2 (EK1501)^BlowerHouse_1 (EK1122)^Term 42 (EK1100)^Term 54 (EL2809)^Channel 10^Output} *)
	STP.B201A3_AirBlowerS1_RunCmd AT %QX14.6 : BOOL;	(*  ~ {LinkedWith:TIID^C6920 (EtherCAT)^ScadaRoom_KouplerUTP (EK1100)^ScadaRoom_KouplerFiber (EK1521)^BlowerHouse_2 (EK1501)^BlowerHouse_1 (EK1122)^Term 42 (EK1100)^Term 54 (EL2809)^Channel 11^Output} *)
	STP.P201A1_DesludgePump_RunCmd AT %QX14.7 : BOOL;	(*  ~ {LinkedWith:TIID^C6920 (EtherCAT)^ScadaRoom_KouplerUTP (EK1100)^ScadaRoom_KouplerFiber (EK1521)^BlowerHouse_2 (EK1501)^BlowerHouse_1 (EK1122)^Term 42 (EK1100)^Term 54 (EL2809)^Channel 12^Output} *)
	STP.P201A2_DesludgePump_RunCmd AT %QX15.0 : BOOL;	(*  ~ {LinkedWith:TIID^C6920 (EtherCAT)^ScadaRoom_KouplerUTP (EK1100)^ScadaRoom_KouplerFiber (EK1521)^BlowerHouse_2 (EK1501)^BlowerHouse_1 (EK1122)^Term 42 (EK1100)^Term 54 (EL2809)^Channel 13^Output} *)
	STP.AUXA1_ReactorS1R1_OpsStat AT %QX15.1 : BOOL;	(*  ~ {LinkedWith:TIID^C6920 (EtherCAT)^ScadaRoom_KouplerUTP (EK1100)^ScadaRoom_KouplerFiber (EK1521)^BlowerHouse_2 (EK1501)^BlowerHouse_1 (EK1122)^Term 42 (EK1100)^Term 55 (EL2809)^Channel 1^Output} *)
	STP.AUXA2_ReactorS1R2_OpsStat AT %QX15.2 : BOOL;	(*  ~ {LinkedWith:TIID^C6920 (EtherCAT)^ScadaRoom_KouplerUTP (EK1100)^ScadaRoom_KouplerFiber (EK1521)^BlowerHouse_2 (EK1501)^BlowerHouse_1 (EK1122)^Term 42 (EK1100)^Term 55 (EL2809)^Channel 2^Output} *)
	STP.AUXA3_ReactorS1R3_OpsStat AT %QX15.3 : BOOL;	(*  ~ {LinkedWith:TIID^C6920 (EtherCAT)^ScadaRoom_KouplerUTP (EK1100)^ScadaRoom_KouplerFiber (EK1521)^BlowerHouse_2 (EK1501)^BlowerHouse_1 (EK1122)^Term 42 (EK1100)^Term 55 (EL2809)^Channel 3^Output} *)
	STP.AUXA4_ReactorS1R4_OpsStat AT %QX15.4 : BOOL;	(*  ~ {LinkedWith:TIID^C6920 (EtherCAT)^ScadaRoom_KouplerUTP (EK1100)^ScadaRoom_KouplerFiber (EK1521)^BlowerHouse_2 (EK1501)^BlowerHouse_1 (EK1122)^Term 42 (EK1100)^Term 55 (EL2809)^Channel 4^Output} *)
	STP.AUXB1_ReactorS2R1_OpsStat AT %QX15.5 : BOOL;	(*  ~ {LinkedWith:TIID^C6920 (EtherCAT)^ScadaRoom_KouplerUTP (EK1100)^ScadaRoom_KouplerFiber (EK1521)^BlowerHouse_2 (EK1501)^BlowerHouse_1 (EK1122)^Term 42 (EK1100)^Term 55 (EL2809)^Channel 5^Output} *)
	STP.AUXB2_ReactorS2R2_OpsStat AT %QX15.6 : BOOL;	(*  ~ {LinkedWith:TIID^C6920 (EtherCAT)^ScadaRoom_KouplerUTP (EK1100)^ScadaRoom_KouplerFiber (EK1521)^BlowerHouse_2 (EK1501)^BlowerHouse_1 (EK1122)^Term 42 (EK1100)^Term 55 (EL2809)^Channel 6^Output} *)
	STP.AUXB3_ReactorS2R3_OpsStat AT %QX15.7 : BOOL;	(*  ~ {LinkedWith:TIID^C6920 (EtherCAT)^ScadaRoom_KouplerUTP (EK1100)^ScadaRoom_KouplerFiber (EK1521)^BlowerHouse_2 (EK1501)^BlowerHouse_1 (EK1122)^Term 42 (EK1100)^Term 55 (EL2809)^Channel 7^Output} *)
	STP.AUXB4_ReactorS2R4_OpsStat AT %QX16.0 : BOOL;	(*  ~ {LinkedWith:TIID^C6920 (EtherCAT)^ScadaRoom_KouplerUTP (EK1100)^ScadaRoom_KouplerFiber (EK1521)^BlowerHouse_2 (EK1501)^BlowerHouse_1 (EK1122)^Term 42 (EK1100)^Term 55 (EL2809)^Channel 8^Output} *)
	STP.AUXA5_BlowerS1R1 AT %QX16.1 : BOOL;	(*  ~ {LinkedWith:TIID^C6920 (EtherCAT)^ScadaRoom_KouplerUTP (EK1100)^ScadaRoom_KouplerFiber (EK1521)^BlowerHouse_2 (EK1501)^BlowerHouse_1 (EK1122)^Term 42 (EK1100)^Term 55 (EL2809)^Channel 9^Output} *)
	STP.AUXA6_BlowerS1R2 AT %QX16.2 : BOOL;	(*  ~ {LinkedWith:TIID^C6920 (EtherCAT)^ScadaRoom_KouplerUTP (EK1100)^ScadaRoom_KouplerFiber (EK1521)^BlowerHouse_2 (EK1501)^BlowerHouse_1 (EK1122)^Term 42 (EK1100)^Term 55 (EL2809)^Channel 10^Output} *)
	STP.AUXA7_BlowerS1R3 AT %QX16.3 : BOOL;	(*  ~ {LinkedWith:TIID^C6920 (EtherCAT)^ScadaRoom_KouplerUTP (EK1100)^ScadaRoom_KouplerFiber (EK1521)^BlowerHouse_2 (EK1501)^BlowerHouse_1 (EK1122)^Term 42 (EK1100)^Term 55 (EL2809)^Channel 11^Output} *)
	STP.AUXB5_BlowerS2R1 AT %QX16.4 : BOOL;	(*  ~ {LinkedWith:TIID^C6920 (EtherCAT)^ScadaRoom_KouplerUTP (EK1100)^ScadaRoom_KouplerFiber (EK1521)^BlowerHouse_2 (EK1501)^BlowerHouse_1 (EK1122)^Term 42 (EK1100)^Term 55 (EL2809)^Channel 12^Output} *)
	STP.AUXB6_BlowerS2R2 AT %QX16.5 : BOOL;	(*  ~ {LinkedWith:TIID^C6920 (EtherCAT)^ScadaRoom_KouplerUTP (EK1100)^ScadaRoom_KouplerFiber (EK1521)^BlowerHouse_2 (EK1501)^BlowerHouse_1 (EK1122)^Term 42 (EK1100)^Term 55 (EL2809)^Channel 13^Output} *)
	STP.AUXB7_BlowerS2R3 AT %QX16.6 : BOOL;	(*  ~ {LinkedWith:TIID^C6920 (EtherCAT)^ScadaRoom_KouplerUTP (EK1100)^ScadaRoom_KouplerFiber (EK1521)^BlowerHouse_2 (EK1501)^BlowerHouse_1 (EK1122)^Term 42 (EK1100)^Term 55 (EL2809)^Channel 14^Output} *)
	STP.AUX201_CommonAlarm AT %QX72.3 : BOOL;	(*  ~ {LinkedWith:TIID^C6920 (EtherCAT)^ScadaRoom_KouplerUTP (EK1100)^ScadaRoom_KouplerFiber (EK1521)^BlowerHouse_2 (EK1501)^BlowerHouse_1 (EK1122)^Term 42 (EK1100)^Term 55 (EL2809)^Channel 15^Output} *)
	STP.AUX202_PLCRunStat AT %QX72.4 : BOOL;	(*  ~ {LinkedWith:TIID^C6920 (EtherCAT)^ScadaRoom_KouplerUTP (EK1100)^ScadaRoom_KouplerFiber (EK1521)^BlowerHouse_2 (EK1501)^BlowerHouse_1 (EK1122)^Term 42 (EK1100)^Term 55 (EL2809)^Channel 16^Output} *)
	STP.TMT03_FanStatus AT %IX49.1 : BOOL;	(*  ~ {LinkedWith:TIID^C6920 (EtherCAT)^ScadaRoom_KouplerUTP (EK1100)^ScadaRoom_KouplerFiber (EK1521)^BlowerHouse_2 (EK1501)^BlowerHouse_1 (EK1122)^Term 42 (EK1100)^Term 43 (EL1809)^Channel 1^Input} *)
	STP.DP03_DoorPanelStatus AT %IX49.2 : BOOL;	(*  ~ {LinkedWith:TIID^C6920 (EtherCAT)^ScadaRoom_KouplerUTP (EK1100)^ScadaRoom_KouplerFiber (EK1521)^BlowerHouse_2 (EK1501)^BlowerHouse_1 (EK1122)^Term 42 (EK1100)^Term 43 (EL1809)^Channel 2^Input} *)
	STP.XV261B_DecanterR1_OverloadStat AT %IX49.3 : BOOL;	(*  ~ {LinkedWith:TIID^C6920 (EtherCAT)^ScadaRoom_KouplerUTP (EK1100)^ScadaRoom_KouplerFiber (EK1521)^BlowerHouse_2 (EK1501)^Term 29 (EL1809)^Channel 3^Input} *)
	STP.XV262B_DecanterR2_OverloadStat AT %IX49.4 : BOOL;	(*  ~ {LinkedWith:TIID^C6920 (EtherCAT)^ScadaRoom_KouplerUTP (EK1100)^ScadaRoom_KouplerFiber (EK1521)^BlowerHouse_2 (EK1501)^Term 29 (EL1809)^Channel 4^Input} *)
	STP.XV263B_DecanterR3_OverloadStat AT %IX49.5 : BOOL;	(*  ~ {LinkedWith:TIID^C6920 (EtherCAT)^ScadaRoom_KouplerUTP (EK1100)^ScadaRoom_KouplerFiber (EK1521)^BlowerHouse_2 (EK1501)^Term 29 (EL1809)^Channel 5^Input} *)
	STP.XV264B_DecanterR4_OverloadStat AT %IX49.6 : BOOL;	(*  ~ {LinkedWith:TIID^C6920 (EtherCAT)^ScadaRoom_KouplerUTP (EK1100)^ScadaRoom_KouplerFiber (EK1521)^BlowerHouse_2 (EK1501)^Term 29 (EL1809)^Channel 6^Input} *)
	STP.M200B1A_MixerR1_RunStat AT %IX49.7 : BOOL;	(*  ~ {LinkedWith:TIID^C6920 (EtherCAT)^ScadaRoom_KouplerUTP (EK1100)^ScadaRoom_KouplerFiber (EK1521)^BlowerHouse_2 (EK1501)^Term 30 (EL1809)^Channel 1^Input} *)
	STP.M200B1B_MixerR1_RunStat AT %IX50.0 : BOOL;	(*  ~ {LinkedWith:TIID^C6920 (EtherCAT)^ScadaRoom_KouplerUTP (EK1100)^ScadaRoom_KouplerFiber (EK1521)^BlowerHouse_2 (EK1501)^Term 30 (EL1809)^Channel 2^Input} *)
	STP.M200B1C_MixerR1_RunStat AT %IX50.1 : BOOL;	(*  ~ {LinkedWith:TIID^C6920 (EtherCAT)^ScadaRoom_KouplerUTP (EK1100)^ScadaRoom_KouplerFiber (EK1521)^BlowerHouse_2 (EK1501)^Term 30 (EL1809)^Channel 3^Input} *)
	STP.M200B2A_MixerR2_RunStat AT %IX50.2 : BOOL;	(*  ~ {LinkedWith:TIID^C6920 (EtherCAT)^ScadaRoom_KouplerUTP (EK1100)^ScadaRoom_KouplerFiber (EK1521)^BlowerHouse_2 (EK1501)^Term 30 (EL1809)^Channel 4^Input} *)
	STP.M200B2B_MixerR2_RunStat AT %IX50.3 : BOOL;	(*  ~ {LinkedWith:TIID^C6920 (EtherCAT)^ScadaRoom_KouplerUTP (EK1100)^ScadaRoom_KouplerFiber (EK1521)^BlowerHouse_2 (EK1501)^Term 30 (EL1809)^Channel 5^Input} *)
	STP.M200B2C_MixerR2_RunStat AT %IX50.4 : BOOL;	(*  ~ {LinkedWith:TIID^C6920 (EtherCAT)^ScadaRoom_KouplerUTP (EK1100)^ScadaRoom_KouplerFiber (EK1521)^BlowerHouse_2 (EK1501)^Term 30 (EL1809)^Channel 6^Input} *)
	STP.M200B3A_MixerR3_RunStat AT %IX50.5 : BOOL;	(*  ~ {LinkedWith:TIID^C6920 (EtherCAT)^ScadaRoom_KouplerUTP (EK1100)^ScadaRoom_KouplerFiber (EK1521)^BlowerHouse_2 (EK1501)^Term 30 (EL1809)^Channel 7^Input} *)
	STP.M200B3B_MixerR3_RunStat AT %IX50.6 : BOOL;	(*  ~ {LinkedWith:TIID^C6920 (EtherCAT)^ScadaRoom_KouplerUTP (EK1100)^ScadaRoom_KouplerFiber (EK1521)^BlowerHouse_2 (EK1501)^Term 30 (EL1809)^Channel 8^Input} *)
	STP.M200B3C_MixerR3_RunStat AT %IX50.7 : BOOL;	(*  ~ {LinkedWith:TIID^C6920 (EtherCAT)^ScadaRoom_KouplerUTP (EK1100)^ScadaRoom_KouplerFiber (EK1521)^BlowerHouse_2 (EK1501)^Term 30 (EL1809)^Channel 9^Input} *)
	STP.M200B4A_MixerR4_RunStat AT %IX51.0 : BOOL;	(*  ~ {LinkedWith:TIID^C6920 (EtherCAT)^ScadaRoom_KouplerUTP (EK1100)^ScadaRoom_KouplerFiber (EK1521)^BlowerHouse_2 (EK1501)^Term 30 (EL1809)^Channel 10^Input} *)
	STP.M200B4B_MixerR4_RunStat AT %IX51.1 : BOOL;	(*  ~ {LinkedWith:TIID^C6920 (EtherCAT)^ScadaRoom_KouplerUTP (EK1100)^ScadaRoom_KouplerFiber (EK1521)^BlowerHouse_2 (EK1501)^Term 30 (EL1809)^Channel 11^Input} *)
	STP.M200B4C_MixerR4_RunStat AT %IX51.2 : BOOL;	(*  ~ {LinkedWith:TIID^C6920 (EtherCAT)^ScadaRoom_KouplerUTP (EK1100)^ScadaRoom_KouplerFiber (EK1521)^BlowerHouse_2 (EK1501)^Term 30 (EL1809)^Channel 12^Input} *)
	STP.B201B1_AirBlowerS2_RunStat AT %IX256.7 : BOOL;	(*  ~ {LinkedWith:TIID^C6920 (EtherCAT)^ScadaRoom_KouplerUTP (EK1100)^ScadaRoom_KouplerFiber (EK1521)^BlowerHouse_2 (EK1501)^Term 30 (EL1809)^Channel 13^Input} *)
